Yaskawa INFORM job: OK_R2_O38-47,64(1)(90,180)OKKR.JBI

/JOB
//NAME OK_R2_O38-47,64(1)(90,180)OKKR
///FOLDERNAME X4
//POS
///NPOS 675,675,675,19,0,0
///TOOL 0
///POSTYPE PULSE
///PULSE
C00000=-90909,-97924,-91406,-33882,56334,85304
C00001=-91259,-96225,-90754,-33542,56592,85046
C00002=-84346,-10282,-49110,5038,88729,85099
C00003=-80520,72534,46153,-179,119568,81737
C00004=-84341,50404,17488,-7249,115666,79799
C00005=-84629,52012,20689,-7225,114506,79766
C00006=-84629,51890,21633,-7182,113865,79809
C00007=-84629,52012,20689,-7225,114506,79766
C00008=-84940,55701,25098,-7229,113667,79705
C00009=-84940,55628,25812,-7200,113194,79735
C00010=-84829,53963,24073,-7195,113413,79762
C00011=-84779,55348,25092,-7189,113502,79775
C00012=-83953,58737,25467,-6224,116924,79977
C00013=-84346,-10282,-49110,5038,88729,85099
C00014=-83106,-20728,-52489,-22212,92643,80661
C00015=-106659,-18282,-50653,-15937,87636,73637
C00016=-135463,84611,26036,-8427,98138,63561
C00017=-134711,78652,30015,-19475,126025,58919
C00018=-134415,83458,36943,-18891,124399,59387
C00019=-134415,83178,37391,-18788,124001,59464
C00020=-134415,82845,37969,-18663,123504,59559
C00021=-134415,83107,37513,-18763,123898,59484
C00022=-133823,86478,41707,-18417,123218,59859
C00023=-133823,86166,42311,-18294,122713,59953
C00024=-134051,84793,40603,-18428,122994,59806
C00025=-133823,86534,41603,-18437,123307,59843
C00026=-130836,86678,38865,-21284,122414,55409
C00027=-135463,84611,26036,-8427,98138,63561
C00028=-106659,-18282,-50653,-15937,87636,73637
C00029=-89310,-122172,-106686,-13361,50676,45199
C00030=-123165,-113898,-119110,19125,43336,-19368
C00031=-123668,-102412,-109547,19577,43467,-19587
C00032=-131184,63359,57441,15233,67840,-18691
C00033=-122068,78147,74274,12505,69533,-15106
C00034=-122051,87849,89370,12875,65325,-15559
C00035=-122051,89227,92048,12969,64408,-15664
C00036=-122316,85057,86118,12868,65923,-15592
C00037=-122667,82911,83414,12880,66527,-15655
C00038=-122667,83831,85320,12946,65844,-15732
C00039=-122426,86931,89254,12983,65000,-15737
C00040=-122963,79390,78884,12845,67528,-15654
C00041=-130632,64185,60223,15235,66493,-18662
C00042=-131662,58983,54996,15425,67212,-18954
C00043=-131668,55339,42428,14901,72880,-18222
C00044=-146861,-92393,-105699,36485,53490,-27620
C00045=-148000,-101656,-114811,36865,54640,-27702
C00046=-148000,-101656,-114811,36865,54640,-27702
C00047=-148000,-101656,-114811,36865,54640,-27702
C00048=-159496,-161049,-136264,30615,73499,-21221
C00049=-103228,-122632,-133352,-7038,92284,-523
C00050=-103228,-122632,-133352,-7038,92284,-523
C00051=-103228,-124480,-131601,-7026,90271,-411
C00052=-103391,-121920,-131082,-6996,91247,-517
C00053=-103853,-115329,-128981,-6922,93290,-780
C00054=-103391,-120798,-132087,-7006,92433,-583
C00055=-104641,-114737,-130152,-6774,94243,-1084
C00056=-104641,-114737,-130152,-6774,94243,-1084
C00057=-104641,-116137,-129119,-6762,92896,-1012
C00058=-104641,-115940,-129279,-6764,93095,-1023
C00059=-105111,-108950,-126961,-6694,95208,-1287
C00060=-104576,-115792,-130426,-6785,93876,-1044
C00061=-103741,-127928,-135528,-6927,90867,-609
C00062=-103741,-127928,-135528,-6927,90867,-609
C00063=-103741,-127928,-135528,-6927,90867,-609
C00064=-103865,-116944,-129962,-6921,93061,-771
C00065=-103865,-118485,-128547,-6909,91408,-679
C00066=-103865,-118011,-129031,-6913,91946,-709
C00067=-104350,-111197,-126797,-6823,94018,-978
C00068=-103645,-119716,-131347,-6963,92509,-670
C00069=-126331,-111187,-127566,-2170,93341,-7936
C00070=-126314,-110675,-127191,-2173,93374,-7931
C00071=-126314,-111741,-126360,-2171,92316,-7913
C00072=-126314,-111248,-126762,-2172,92816,-7922
C00073=-126152,-104604,-124481,-2216,94828,-7909
C00074=-126314,-111061,-126906,-2173,93001,-7925
C00075=-125902,-111149,-126935,-2263,92984,-7794
C00076=-132196,-109284,-126305,2386,93568,-14490
C00077=-132014,-110397,-125220,2342,92324,-14457
C00078=-132014,-111538,-124094,2340,91046,-14481
C00079=-132014,-110972,-124684,2340,91699,-14468
C00080=-131346,-109003,-124013,2196,92280,-14246
C00081=-132122,-112463,-125993,2364,91740,-14502
C00082=-130696,-128652,-136015,2037,89553,-14081
C00083=-130696,-128652,-136015,2037,89553,-14081
C00084=-134573,-129962,-127961,2886,84044,-15460
C00085=-135247,-123905,-124729,3029,85191,-15657
C00086=-135247,-124242,-122895,3032,83891,-15687
C00087=-135059,-121526,-122583,2986,85086,-15595
C00088=-134621,-115318,-120572,2888,87018,-15405
C00089=-135273,-124345,-124575,3033,84868,-15671
C00090=-101634,-140552,-130463,-4330,80438,-4385
C00091=-100831,-135445,-127742,-4507,81431,-4148
C00092=-100831,-135220,-126147,-4516,80567,-4118
C00093=-100831,-135304,-126661,-4513,80840,-4129
C00094=-101541,-127818,-124438,-4340,83274,-4455
C00095=-100689,-136992,-128168,-4541,80909,-4084
C00096=-101700,-117063,-135109,-4321,95328,-4920
C00097=-101700,-117063,-135109,-4321,95328,-4920
C00098=-107464,-106510,-121453,-3057,92107,-6652
C00099=-105693,-105772,-119256,-3437,91202,-6062
C00100=-105693,-106748,-117862,-3435,89847,-6024
C00101=-105693,-106325,-118509,-3436,90460,-6041
C00102=-104724,-99451,-116018,-3652,92493,-5788
C00103=-105563,-106984,-120499,-3466,91350,-6023
C00104=-97637,-124436,-133710,-5150,90918,-3458
C00105=-101700,-117063,-135109,-4321,95328,-4920
C00106=-101700,-117063,-135109,-4321,95328,-4920
C00107=-113885,-115939,-123860,-1658,88568,-8649
C00108=-113885,-115976,-123799,-1658,88510,-8649
C00109=-113885,-116503,-122835,-1658,87648,-8639
C00110=-113928,-115223,-122529,-1647,88114,-8658
C00111=-114061,-111130,-121156,-1620,89368,-8717
C00112=-113613,-117192,-124203,-1715,88138,-8556
C00113=-77135,-109099,-124316,-9289,94737,2930
C00114=-77964,-100968,-118468,-9143,95217,2626
C00115=-77964,-101677,-117713,-9127,94398,2685
C00116=-77964,-101560,-117850,-9129,94540,2675
C00117=-78928,-97543,-116360,-8967,95572,2290
C00118=-77908,-100245,-119438,-9173,96179,2574
C00119=-71973,-123086,-130703,-10190,92110,4818
C00120=-61369,-106979,-129386,18745,110548,-43775
C00121=-54050,-118433,-122678,29834,105379,-66043
C00122=-54050,-118432,-122677,29849,105379,-66042
C00123=-52380,-128849,-120518,29019,98947,-67079
C00124=-52380,-128559,-118965,28945,98241,-67262
C00125=-52380,-128751,-119946,28990,98681,-67146
C00126=-50245,-132811,-121152,28917,96763,-66805
C00127=-52380,-128751,-119946,28990,98681,-67146
C00128=-49374,-119498,-117890,29381,100712,-65454
C00129=-49135,-119946,-117683,29342,100317,-65463
C00130=-49135,-119959,-116418,29258,99629,-65643
C00131=-49135,-119963,-116925,29289,99902,-65571
C00132=-47420,-122909,-117861,29192,98489,-65269
C00133=-49767,-118756,-118042,29437,101266,-65461
C00134=-58824,-127197,-127906,29549,105900,-67783
C00135=-58824,-127197,-127906,29549,105900,-67783
C00136=-55789,-138532,-125635,28743,98511,-68512
C00137=-54845,-137144,-123724,28738,97781,-68329
C00138=-54845,-136558,-122036,28679,97131,-68490
C00139=-54845,-136878,-122937,28709,97474,-68406
C00140=-52687,-141381,-124200,28678,95380,-68093
C00141=-56052,-135036,-125386,28893,100051,-68223
C00142=-56052,-135036,-125386,28893,100051,-68223
C00143=-54923,-136926,-123517,28734,97796,-68355
C00144=-54923,-136449,-122129,28684,97260,-68488
C00145=-54923,-136715,-122887,28711,97551,-68416
C00146=-52628,-141500,-124230,28677,95326,-68085
C00147=-54923,-138669,-131970,29176,101590,-67387
C00148=-49576,-128334,-132403,27234,106270,-69223
C00149=-44922,-139442,-128392,26353,97465,-69516
C00150=-43106,-142181,-127565,26251,95168,-69348
C00151=-43106,-141292,-125343,26201,94348,-69532
C00152=-43106,-141708,-126356,26223,94717,-69449
C00153=-42222,-150085,-128620,26118,91814,-69764
C00154=-43106,-141708,-126356,26223,94717,-69449
C00155=-58006,-149727,-131155,24086,101568,-78058
C00156=-67130,-160484,-130477,19696,102779,-86761
C00157=-65656,-163702,-131169,20680,100336,-85246
C00158=-25743,-109032,-115433,27145,106620,-70118
C00159=-31386,-185321,-134069,30256,67850,-60806
C00160=-40913,-181249,-136978,30366,76641,-63974
C00161=-31337,-124593,-132531,25311,107075,-53461
C00162=-107165,-96970,-126665,-3187,100215,-6761
C00163=-107165,-106401,-121090,-3121,91950,-6553
C00164=-99006,-123912,-120398,-10471,76789,317
C00165=-104449,-120133,-119195,-8811,77334,-1598
C00166=-136314,-76901,-102772,1273,87959,-12257
C00167=-129245,-75238,-102051,-6216,89043,-4909
C00168=-138081,-104464,-122106,1833,85725,-12838
C00169=-119260,-105046,-123410,-8534,87528,-2432
C00170=-124620,-151805,-134891,-7305,72242,-3267
C00171=-124614,-151414,-134787,-7302,72378,-3273
C00172=-124612,-151215,-134734,-7300,72449,-3276
C00173=-124620,-151805,-134891,-7305,72242,-3267
C00174=-127969,-108981,-129625,-6073,90620,-5362
C00175=-128058,-112032,-130642,-6044,89675,-5344
C00176=-99990,-117497,-120264,-13536,83880,4252
C00177=-95946,-115412,-117807,-14495,84133,5598
C00178=-139069,-101671,-113062,-2900,83618,-8638
C00179=-134512,-124069,-125019,-4259,79673,-7022
C00180=-124704,-125859,-130096,-7035,82535,-3892
C00181=-99313,-127153,-133045,12119,95446,-32872
C00182=-57886,-133831,-130402,29291,103936,-67934
C00183=-55789,-138532,-125635,28743,98511,-68512
C00184=-48693,-117877,-116324,29063,104784,-69163
C00185=-50073,-120833,-117390,28223,106210,-71565
C00186=-68626,-163926,-129258,19114,104295,-87122
C00187=-70376,-133538,-127464,20847,118406,-85282
C00188=-70376,-133538,-127464,20847,118406,-85282
C00189=-57461,-97931,-109353,30188,105270,-63675
C00190=-56121,-79134,-101591,31100,116741,-68778
C00191=-90239,-137211,-122130,21625,111934,-84005
C00192=-78206,-119593,-116830,16675,122083,-90308
C00193=-77714,-101700,-117389,19308,131076,-88387
C00194=-81561,-124200,-134149,21063,125175,-90603
C00195=-103376,-109759,-132308,-3968,97270,-5504
C00196=-101634,-140552,-130463,-4330,80438,-4385
C00197=-110031,-125673,-123303,3182,83425,-15942
C00198=-90641,-116743,-120449,-11075,89773,6751
C00199=-125358,-116095,-120243,-4332,86705,-4548
C00200=-114606,-95150,-113030,-13927,98680,11559
C00201=-109678,-119625,-133746,-14623,99658,13079
C00202=-112326,-124641,-135293,-14185,97639,12436
C00203=-113675,-111285,-124420,-14007,97585,11993
C00204=-113699,-111426,-124467,-14002,97539,11990
C00205=-124004,-129907,-130136,-8507,87303,2218
C00206=-139409,-131326,-130615,456,84743,-11777
C00207=-149006,-99791,-120232,2566,94725,-14751
C00208=-149042,-99754,-120218,2574,94737,-14762
C00209=-144445,-99331,-120062,1565,94748,-13320
C00210=-148134,-92536,-117492,2386,96740,-14437
C00211=-154718,-145008,-134516,3815,80522,-16974
C00212=-155631,-143491,-134098,4008,81086,-17267
C00213=-124045,-119827,-121338,-6126,86009,-1689
C00214=-127884,-116949,-120404,-5328,86643,-2988
C00215=-148100,-95243,-112662,-980,92257,-9671
C00216=-137287,-91556,-109748,-13625,92659,296
C00217=-127829,-127486,-128792,-15513,87749,4031
C00218=-127829,-122446,-134816,-15592,93826,3264
C00219=-125285,-108995,-105645,24533,66859,-22374
C00220=-121876,-100663,-100590,22961,66967,-21017
C00221=-120611,-97454,-98556,22372,66992,-20522
C00222=-120728,-95778,-96365,22498,66572,-20652
C00223=-120611,-97454,-98556,22372,66992,-20522
C00224=-120972,-98646,-98782,22597,66650,-20731
C00225=-119814,-94892,-97816,21908,67582,-20099
C00226=-120972,-98646,-98782,22597,66650,-20731
C00227=-122255,-101873,-100811,23195,66623,-21236
C00228=-125713,-110249,-105850,24792,66512,-22621
C00229=-125414,-109454,-110952,25434,70557,-21724
C00230=-121886,-100912,-105844,23885,70668,-20357
C00231=-120575,-97642,-103795,23303,70688,-19860
C00232=-120636,-96154,-101667,23400,70203,-19982
C00233=-120575,-97642,-103795,23303,70688,-19860
C00234=-121028,-97980,-103315,23548,70382,-20093
C00235=-119871,-93906,-102218,22897,71374,-19458
C00236=-121028,-97980,-103315,23548,70382,-20093
C00237=-122351,-101230,-105354,24132,70373,-20595
C00238=-125908,-109706,-110431,25687,70298,-21973
C00239=-125468,-108852,-114009,26132,73198,-21211
C00240=-121864,-100250,-108878,24604,73277,-19846
C00241=-120523,-96969,-106822,24029,73283,-19350
C00242=-120543,-95651,-104748,24106,72739,-19471
C00243=-120523,-96969,-106822,24029,73283,-19350
C00244=-121096,-97384,-106424,24308,73024,-19616
C00245=-119937,-93066,-105230,23683,74062,-18974
C00246=-121096,-97384,-106424,24308,73024,-19616
C00247=-122450,-100644,-108468,24886,73032,-20117
C00248=-126090,-109173,-113564,26418,72994,-21493
C00249=-126107,-105383,-120588,25792,78658,-20214
C00250=-115870,-101424,-121533,-41206,90180,-3452
C00251=-115851,-106682,-115012,-41260,85065,-1433
C00252=-119242,-98694,-109765,-40357,84214,-2540
C00253=-120508,-95652,-107669,-40003,83867,-2939
C00254=-120512,-93942,-105232,-40036,83383,-2757
C00255=-120508,-95652,-107669,-40003,83867,-2939
C00256=-119976,-95300,-106376,-40178,83625,-2624
C00257=-123146,-93912,-105979,-39274,82602,-3565
C00258=-119976,-95300,-106376,-40178,83625,-2624
C00259=-118706,-98291,-108457,-40527,83992,-2228
C00260=-115305,-106116,-113657,-41413,84900,-1133
C00261=-117529,-113204,-110114,-15038,59483,16836
C00262=-119860,-102582,-104476,-13511,61010,15725
C00263=-120710,-98611,-102232,-12973,61516,15338
C00264=-120712,-96036,-99318,-13028,61058,15391
C00265=-120710,-98611,-102232,-12973,61516,15338
C00266=-120133,-97446,-101425,-13271,61707,15536
C00267=-121539,-92419,-99938,-12330,63118,14842
C00268=-120133,-97446,-101425,-13271,61707,15536
C00269=-119274,-101350,-103659,-13810,61233,15923
C00270=-116924,-111770,-109266,-15331,59803,17031
C00271=-118012,-90030,-113480,-10859,76824,11039
C00272=-121151,-43618,-104634,1145,105190,-4571
C00273=-120753,-40362,-99446,1000,103667,-4481
C00274=-120604,-39041,-97355,946,103057,-4446
C00275=-120606,-40163,-95662,941,101440,-4458
C00276=-120604,-39041,-97355,946,103057,-4446
C00277=-120772,-35445,-95769,1008,103931,-4483
C00278=-120462,-29091,-92658,908,105279,-4391
C00279=-120772,-35445,-95769,1008,103931,-4483
C00280=-120921,-36668,-97839,1062,104577,-4517
C00281=-121319,-39651,-102962,1210,106200,-4605
C00282=-108629,-121399,-122702,-16889,67135,14241
C00283=-115336,-113367,-105488,-19088,53546,18271
C00284=-117865,-102996,-100223,-17109,54980,16930
C00285=-118786,-99066,-98108,-16412,55481,16461
C00286=-118815,-96798,-95161,-16518,54853,16552
C00287=-118786,-99066,-98108,-16412,55481,16461
C00288=-119112,-97264,-98148,-16039,56331,16193
C00289=-118757,-93015,-97035,-15990,57843,16106
C00290=-119112,-97264,-98148,-16039,56331,16193
C00291=-123316,-98367,-98161,-13561,55035,14648
C00292=-126858,-97217,-97820,-11275,54872,13210
C00293=-123316,-98367,-98161,-13561,55035,14648
C00294=-122519,-102389,-100318,-14180,54451,15058
C00295=-120328,-113051,-105701,-15959,52759,16243
C00296=-124093,-110707,-95637,16539,52225,-18162
C00297=-121727,-101468,-90458,14864,53273,-16967
C00298=-120864,-97923,-88367,14268,53637,-16545
C00299=-120864,-95769,-85768,14357,53158,-16613
C00300=-120864,-97923,-88367,14268,53637,-16545
C00301=-120753,-94948,-87925,13988,54838,-16331
C00302=-119636,-91806,-87160,13170,55764,-15745
C00303=-120753,-94948,-87925,13988,54838,-16331
C00304=-121593,-98445,-90034,14553,54501,-16732
C00305=-123889,-107558,-95262,16133,53518,-17861
C00306=-123907,-109460,-104253,15319,57915,-17198
C00307=-120718,-89127,-94408,-93,103364,81793
C00308=-120702,-88967,-86044,-90,98299,81802
C00309=-120714,-92346,-83648,-90,95088,81800
C00310=-120719,-93530,-82604,-90,93837,81800
C00311=-120721,-91291,-79709,-90,93204,81799
C00312=-120719,-93530,-82604,-90,93837,81800
C00313=-120503,-94372,-82680,-81,93451,81873
C00314=-120503,-97134,-83277,-81,92401,81874
C00315=-120503,-94372,-82680,-81,93451,81873
C00316=-120501,-93212,-83739,-81,94699,81873
C00317=-120496,-89894,-86173,-82,97902,81873
C00318=-120512,-90208,-94601,-84,102927,81864
C00319=-120739,-87258,-85833,-92,99047,81789
C00320=-120752,-90752,-83510,-91,95822,81787
C00321=-120758,-91982,-82493,-91,94564,81786
C00322=-120759,-89478,-79257,-91,93861,81786
C00323=-120758,-91982,-82493,-91,94564,81786
C00324=-120462,-95334,-83503,-80,93464,81887
C00325=-120461,-97919,-84058,-79,92477,81888
C00326=-120462,-95334,-83503,-80,93464,81887
C00327=-120460,-94163,-84562,-80,94717,81887
C00328=-120456,-90813,-86994,-80,97935,81887
C00329=-121033,-93279,-128320,140,99068,-4698
C00330=-120997,-110061,-117241,128,83627,-4703
C00331=-120579,-101211,-110995,15,84330,-4566
C00332=-120424,-97983,-108548,-25,84483,-4515
C00333=-120430,-96385,-106046,-24,83763,-4517
C00334=-120424,-97983,-108548,-25,84483,-4515
C00335=-120936,-92390,-106244,111,85940,-4681
C00336=-120538,-86818,-104536,4,87751,-4552
C00337=-120936,-92390,-106244,111,85940,-4681
C00338=-121096,-95373,-108656,154,85891,-4732
C00339=-121527,-103462,-114785,270,85508,-4872
C00340=-75677,-91018,-121004,-38809,104477,-3256
C00341=-86494,-89564,-122641,-29897,102391,-4704
C00342=-121241,-108971,-117698,1136,79653,-4828
C00343=-120728,-99263,-111358,963,80734,-4651
C00344=-120539,-95742,-108880,900,81016,-4587
C00345=-120543,-94296,-106552,902,80326,-4593
C00346=-120539,-95742,-108880,900,81016,-4587
C00347=-120728,-93992,-107595,961,81127,-4647
C00348=-120728,-90301,-106424,959,82303,-4638
C00349=-120728,-93992,-107595,961,81127,-4647
C00350=-121024,-97533,-112143,1058,82109,-4735
C00351=-121551,-107098,-118478,1235,81100,-4915
C00352=-121569,-100080,-124444,1231,88376,-4850
C00353=-117898,-83225,-110918,-12916,113641,67504
C00354=-119870,-90654,-110250,-12481,109228,67312
C00355=-120686,-93336,-109842,-12338,107519,67211
C00356=-120688,-92183,-107571,-12276,106730,67294
C00357=-120686,-93336,-109842,-12338,107519,67211
C00358=-120163,-91649,-109473,-12395,108219,67318
C00359=-121681,-97188,-111137,-12239,106219,67001
C00360=-120163,-91649,-109473,-12395,108219,67318
C00361=-119359,-88923,-109851,-12543,109932,67413
C00362=-117416,-81399,-110449,-12994,114344,67589
C00363=-120617,-94125,-108136,8857,121741,88541
C00364=-120616,-94449,-107526,8800,121205,88496
C00365=-136098,-107181,-107429,16269,112846,84409
C00366=-120444,-95183,-107742,8816,120947,88541
C00367=-119761,-91680,-105499,9024,121288,-74873
C00368=-120616,-95784,-105179,-19399,105655,65758
C00369=-120617,-94769,-108163,-19676,107886,65380
C00370=-121686,-93853,-106574,-24019,104588,57765
C00371=-120617,-92780,-110041,-24421,107344,57569
C00372=-120617,-90665,-112384,-24828,109654,57058
C00373=-120619,-82046,-117525,-26421,116533,55408
C00374=-120645,-81988,-112872,-3577,88664,15070
C00375=-120614,-96077,-90479,12976,48732,-14983
C00376=-120612,-93911,-81283,13967,44304,-15634
C00377=-120612,-93390,-79613,14157,43566,-15753
C00378=-121252,-93346,-79166,14714,43437,-16096
C00379=-121500,-95247,-79374,15137,42660,-16355
C00380=-120782,-94947,-80724,14317,43483,-15851
C00381=-120611,-93982,-79716,14233,43318,-15795
C00382=-120612,-95725,-83890,13821,44941,-15536
C00383=-121326,-94847,-83951,14224,45559,-15784
C00384=-120613,-94980,-84633,13612,45776,-15407
C00385=-120613,-95388,-86250,13438,46540,-15293
C00386=-120616,-96933,-104006,-5046,49827,-739
C00387=-120616,-97132,-103061,-5097,49146,-704
C00388=-120617,-95323,-101728,-5088,49256,-711
C00389=-120871,-100699,-104338,-4972,48087,-759
C00390=-120795,-98262,-101888,-5054,47837,-712
C00391=-120618,-95198,-103493,-5003,50401,-770
C00392=-121122,-95129,-103646,-4600,50501,-986
C00393=-120617,-97030,-104927,-5009,50342,-766
C00394=-120617,-96757,-105844,-4959,51045,-801
C00395=-120618,-92718,-112658,-4589,57292,-1090
C00396=-108098,-105677,-132023,-7461,89264,328
C00397=-80455,-75739,-120669,-16714,100968,7375
C00398=-97258,-84752,-105297,-10869,90674,3530
C00399=-97358,-86422,-102930,-10833,88387,3696
C00400=-97424,-86715,-102018,-10818,87679,3736
C00401=-97216,-90521,-102980,-10875,86365,3919
C00402=-97404,-84940,-102216,-10822,88698,3655
C00403=-120617,-94266,-106774,-4665,84598,-3614
C00404=-111454,-84543,-103018,-13521,90962,7073
C00405=-109783,-86139,-104921,-12729,90791,5985
C00406=-106092,-100123,-116923,-13597,91547,7106
C00407=-102052,-116072,-128299,-14497,91044,8487
C00408=-91007,-121504,-125767,-15485,91359,21712
C00409=-120613,-95050,-86060,-3557,95049,80550
C00410=-120612,-93945,-81838,-3544,93023,80607
C00411=-121155,-91942,-79314,-3616,92478,80448
C00412=-120652,-94806,-81837,-3543,92579,80606
C00413=-120610,-90975,-79567,-3544,93151,80605
C00414=-150255,-82598,-75582,-4413,93505,70504
C00415=-122384,-91795,-77981,-11848,92227,69969
C00416=-120612,-93489,-79991,-12120,92904,70125
C00417=-120613,-94640,-84016,-12161,94749,69944
C00418=-120614,-96377,-93023,-12320,99298,69491
C00419=-120644,-125570,-121052,6784,67869,5403
C00420=-120615,-96622,-98748,12572,58745,-14095
C00421=-120615,-96643,-96984,12717,57674,-14222
C00422=-127606,-89142,-93330,20657,62312,-19456
C00423=-120926,-99715,-97034,13118,56212,-14526
C00424=-120613,-97817,-97899,12721,57634,-14225
C00425=-120615,-96818,-95655,-6616,54391,-866
C00426=-120615,-97044,-96976,-6561,55085,-910
C00427=-112093,-90513,-93108,-22044,58833,17349
C00428=-120615,-96644,-96112,-9528,53512,9485
C00429=-120615,-96653,-97679,-9416,54459,9397
C00430=-120616,-95373,-105489,-8868,59856,8934
C00431=-117333,-91440,-108817,-14098,83709,30265
C00432=-112347,-94381,-87846,-22750,99580,64599
C00433=-112329,-92021,-78548,-22454,95406,65402
C00434=-115628,-91274,-75119,-22621,92902,64661
C00435=-117255,-90241,-73175,-22718,91835,64269
C00436=-117028,-88603,-73220,-22719,92705,64185
C00437=-116923,-92272,-75451,-22697,92259,64308
C00438=-120553,-90828,-77383,15099,94128,70510
C00439=-120613,-90885,-77384,15804,94030,70628
C00440=-123770,-105111,-82751,16580,84167,79857
C00441=-124886,-104010,-85216,16560,86394,79763
C00442=-120613,-94284,-84162,15892,96365,70931
C00443=-120614,-95920,-93129,16139,100869,71526
C00444=-120649,-92160,-111225,3199,84919,49711
C00445=-120616,-97604,-99172,-11891,40402,23254
C00446=-120614,-96911,-90603,-13253,35598,24030
C00447=-120614,-96763,-89737,-13401,35153,24111
C00448=-121291,-96342,-89250,-12683,34963,23744
C00449=-119113,-97762,-90324,-15090,35268,24978
C00450=-120705,-99580,-90146,-13704,33974,24279
C00451=-121588,-95238,-86691,-12692,33949,23762
C00452=-127502,-77730,-88040,1756,56127,19882
C00453=-125086,-93679,-98074,150,54079,20822
C00454=-120613,-95818,-85653,-14108,33181,24494
C00455=-120615,-97479,-97669,-6545,55280,-923
C00456=-121580,-96410,-96097,-5967,54791,-1285
C00457=-120928,-100587,-97757,-6468,53722,-953
C00458=-120613,-98670,-98620,-6548,55254,-920
C00459=-120615,-96854,-96360,-6584,54805,-893
C00460=-120615,-97074,-97513,-6537,55399,-931
C00461=-114077,-92170,-94328,-19163,57465,15491
C00462=-120615,-97626,-97578,-9481,53904,9448
C00463=-120636,-112691,-117418,-8831,59265,10492
C00464=-120617,-94408,-109491,-7961,65698,13071
C00465=-120616,-97035,-102174,-8375,59902,13490
C00466=-120616,-97254,-100452,-8474,58742,13580
C00467=-120616,-96110,-99125,-8495,58514,13598
C00468=-120614,-98453,-101360,-8481,58685,13585
C00469=-119727,-100186,-100479,-9138,57364,14041
C00470=-120617,-96158,-99373,-8483,58642,13587
C00471=-120616,-97215,-100721,-8458,58926,13566
C00472=-120616,-96978,-102436,-8360,60091,13476
C00473=-120617,-94247,-109716,-7948,65917,13056
C00474=-120616,-96445,-103082,5252,59171,-13430
C00475=-120615,-96888,-94956,5569,53965,-13694
C00476=-120614,-96711,-93127,5642,52935,-13750
C00477=-120614,-96618,-92386,5672,52529,-13773
C00478=-119756,-94067,-91753,5051,53390,-13370
C00479=-120525,-97964,-94062,5589,52861,-13717
C00480=-120614,-96681,-92800,5656,52750,-13760
C00481=-120614,-96709,-92988,5648,52851,-13755
C00482=-120614,-96767,-93400,5632,53074,-13742
C00483=-120614,-96843,-94134,5603,53484,-13720
C00484=-120615,-96977,-95945,5531,54526,-13664
C00485=-120616,-97003,-101109,6851,58481,-13557
C00486=-120615,-97139,-99377,6934,57353,-13629
C00487=-120615,-97164,-98672,6968,56909,-13657
C00488=-119756,-94335,-97933,6375,57832,-13263
C00489=-120570,-98373,-100300,6912,57283,-13615
C00490=-120615,-97165,-99156,6946,57204,-13638
C00491=-120616,-97129,-99856,6912,57651,-13610
C00492=-120616,-96964,-101578,6829,58787,-13537
C00493=-120617,-96349,-105255,7716,61917,-13386
C00494=-120616,-96771,-103611,7804,60699,-13471
C00495=-120616,-96905,-102940,7840,60222,-13505
C00496=-119756,-93851,-102113,7266,61195,-13116
C00497=-120602,-97980,-104523,7800,60639,-13470
C00498=-120616,-96844,-103353,7819,60505,-13485
C00499=-120616,-96699,-104019,7783,60985,-13451
C00500=-120617,-96245,-105652,7696,62212,-13366
C00501=-120618,-92150,-112439,7334,68442,-12961
C00502=-130920,-122289,-127601,-23263,76296,33617
C00503=-126647,-121486,-124764,-14921,71090,19914
C00504=-118673,-117816,-113052,-9081,54805,1270
C00505=-119719,-97166,-102733,-8035,58912,525
C00506=-118944,-92090,-109805,-27006,83902,36269
C00507=-120616,-93914,-111601,-26462,83549,35758
C00508=-120617,-94475,-108119,-24525,75199,30020
C00509=-120618,-90011,-113520,-23738,94905,43572
C00510=-120617,-93534,-109718,-22404,79768,31867
C00511=-120617,-93028,-110386,-24696,84592,28860
C00512=-120617,-93859,-109223,-24523,82429,27907
C00513=-120617,-95217,-106728,-22357,73913,21133
C00514=-120616,-96198,-104144,-16550,64688,11231
C00515=-120616,-97587,-102867,-7505,58697,196
C00516=-120615,-98378,-102979,677,57412,-8649
C00517=-120615,-98092,-104435,2505,58558,-10610
C00518=-120615,-97859,-104607,2041,58746,-10113
C00519=-120615,-97689,-104685,1580,58853,-9618
C00520=-120615,-97267,-104663,-2078,59079,-5700
C00521=-122185,-96113,-104438,-1107,59504,-6297
C00522=-124417,-94235,-103728,259,60020,-7133
C00523=-120617,-96195,-105273,-2057,60007,-5718
C00524=-120617,-95777,-106468,-2039,60956,-5736
C00525=-120690,-30346,-78642,22937,64170,-21118
C00526=-120690,-30346,-78642,22937,64170,-21118
C00527=-98469,-5770,-79404,6171,73775,-13621
C00528=-73961,-64832,-115099,-11040,66386,-6438
C00529=-152983,-151482,-105999,63266,53723,19798
C00530=-133395,-32083,-56059,41211,61963,37621
C00531=-138234,23065,45169,67508,45202,44915
C00532=-136781,30072,55747,70235,43147,43411
C00533=-136213,33214,60449,71542,42329,42699
C00534=-136213,31591,57334,70422,42710,43384
C00535=-136788,30891,57778,71075,42855,42892
C00536=-134893,29619,56778,71118,41623,43172
C00537=-133284,25640,52793,70642,40733,43707
C00538=-131869,22445,49655,70246,39929,44150
C00539=-132436,19576,45433,69035,40713,44782
C00540=-133889,13007,35719,66469,42691,46136
C00541=-120930,8852,32410,71146,24358,44597
C00542=-120056,16713,42856,76185,23038,42237
C00543=-120570,20810,47735,78353,23157,41125
C00544=-120179,17981,45384,78314,22894,41190
C00545=-119718,18730,44666,76295,22791,42223
C00546=-125399,29317,56132,80433,26238,39500
C00547=-125034,24898,50699,78244,26224,40637
C00548=-126001,16678,39521,73266,27604,43020
C00549=-110893,28996,24386,6920,61269,70362
C00550=-121937,-147756,-98721,13314,47766,64479
C00551=-71720,-152863,-104081,-12596,70757,83485
C00552=-71720,-152863,-104081,-12596,70757,83485
C00553=-91982,-28216,-51992,2303,92813,79298
C00554=-105745,54824,-16277,12342,106777,76346
C00555=-79811,47197,33770,-5226,114025,80115
C00556=-80023,42119,31306,-5246,112923,80086
C00557=-80397,41231,31844,-5317,112121,79984
C00558=-80109,39795,28796,-5290,113266,80037
C00559=-80112,42618,33014,-5241,112126,80089
C00560=-81014,41143,31800,-5517,112061,79755
C00561=-81200,40698,29696,-5625,113108,79635
C00562=-82013,41869,30925,-5879,112897,79339
C00563=-84094,42448,33219,-3257,112240,82331
C00564=-82696,41301,31992,-6274,111848,78881
C00565=-83189,43833,33118,-6256,112463,78920
C00566=-80599,47195,33767,-5484,113974,79819
C00567=-80608,45992,24153,-5781,119246,79546
C00568=-80156,46426,18785,-6968,101557,41119
C00569=-78753,47274,23775,-10662,32517,-78562
C00570=-79428,-41610,-51646,-9616,33163,-79071
C00571=-79413,-40970,-42943,-11157,28217,-78271
C00572=-79779,-35257,-36372,-11029,27079,-78324
C00573=-80609,-32957,-33621,-9964,26475,-78835
C00574=-79917,-33213,-35108,-10725,27328,-78472
C00575=-79914,-35155,-35130,-11097,26361,-78286
C00576=-81360,-33165,-33796,-8816,26388,-79388
C00577=-81501,-33436,-35517,-8333,27283,-79626
C00578=-82704,-33725,-35707,-6541,27141,-80488
C00579=-82488,-32797,-33501,-7076,26287,-80226
C00580=-83572,-32639,-33468,-5384,26265,-81042
C00581=-83984,-33203,-37030,-4447,28135,-81499
C00582=-80764,-40975,-42948,-9214,28047,-79206
C00583=-80778,-41615,-51650,-7929,33019,-79872
C00584=-83330,-46575,-52890,-13958,55049,-41505
C00585=-86193,-52033,-54165,-20785,79907,1804
C00586=-87571,-35325,-52921,-25788,81678,348
C00587=-87508,-34952,-39783,-27132,74543,196
C00588=-104644,32154,27534,4448,60513,72731
C00589=-93805,201,18674,23355,11914,69008
C00590=-93808,216,18686,23365,11915,69004
C00591=-93810,222,18691,23369,11915,69002
C00592=-93638,2355,20486,22861,11860,69245
C00593=-93955,-2017,16089,22978,12371,69170
C00594=-93808,210,18682,23363,11914,69005
C00595=-93806,198,18671,23357,11914,69008
C00596=-93804,186,18662,23351,11913,69011
C00597=-93802,180,18657,23347,11913,69012
C00598=-93799,166,18644,23338,11912,69017
C00599=-93810,232,18700,23265,11906,69051
C00600=-93813,246,18712,23275,11907,69047
C00601=-94451,684,18996,25087,12134,68175
C00602=-93990,-1863,16961,23823,11950,68785
C00603=-93814,-607,16661,21825,12670,69707
C00604=-100120,3293,21094,39224,14315,61321
C00605=-100936,-4761,10472,35572,16592,62958
C00606=-101724,-18723,-6868,31140,19848,65000
C00607=-104644,32154,27534,4448,60513,72731
C00608=-81813,-56841,-53371,-53266,50302,14082
C00609=-60380,-131230,-84967,-114894,34586,40161
C00610=-75788,-111312,-115723,-41491,75595,63087
C00611=-90161,-54224,-109841,7916,106787,80704
C00612=-89492,4607,-58591,7657,105439,80800
C00613=-89900,18802,-35938,9766,95357,80687
C00614=-83481,65005,13429,-9056,119285,78997
C00615=-83912,59570,13434,-8836,116477,79073
C00616=-105122,63991,30490,2309,126100,76457
C00617=-105343,61862,26796,2259,127285,76391
C00618=-85790,59910,13822,-8992,116222,78417
C00619=-84859,64061,16437,-8959,116837,78702
C00620=-84733,23156,-31643,-6898,102580,79911
C00621=-89806,-37631,-52942,13196,44828,72538
C00622=-94750,-32934,-45091,18174,44929,69862
C00623=-94750,-25149,-34817,18936,42722,69385
C00624=-107305,-33153,-35053,31246,31625,63156
C00625=-107702,-34958,-34985,32523,30946,62498
C00626=-97165,-24114,-34089,20969,43382,68305
C00627=-95242,-30076,-40811,18964,43932,69406
C00628=-95187,-81119,-79791,20309,40550,69551
C00629=-106636,9561,-40732,-8334,61658,77698
C00630=-105745,52807,-15764,12246,105454,76208
C00631=-120157,82254,53851,-8462,118881,68276
C00632=-120764,76019,49190,-8631,118486,68068
C00633=-120545,73220,47168,-8543,118319,68170
C00634=-121013,73553,46157,-8768,119052,67924
C00635=-120677,76096,50452,-8536,117766,68159
C00636=-121226,74586,48871,-8734,117906,67937
C00637=-121277,74331,46343,-8885,119308,67802
C00638=-123087,79936,53120,-9346,117831,67212
C00639=-123276,78435,53420,-9313,116866,67221
C00640=-123824,79710,55035,-9457,116468,67043
C00641=-123162,86054,59807,-9277,116864,67267
C00642=-123114,53430,10385,-1251,116221,68203
C00643=-136323,52272,9545,44589,64919,61463
C00644=-139783,-33179,-13184,69240,48192,46182
C00645=-137611,-28365,-6875,70201,46216,45730
C00646=-136958,-25590,-3634,70647,45579,45500
C00647=-136770,-25555,-2359,71345,45178,45070
C00648=-137559,-27867,-5282,70853,45921,45309
C00649=-131841,-32953,-8633,70743,41902,45928
C00650=-131975,-36416,-12130,70369,42121,46140
C00651=-134147,-41542,-18435,69427,44030,46529
C00652=-141128,-29133,-31085,43489,44991,50173
C00653=-145944,-19375,-16364,60085,47488,49165
C00654=-146184,-15082,-11889,60605,47355,48817
C00655=-146072,-18893,-14822,60688,47208,48761
C00656=-145286,-17068,-12207,60970,46372,48581
C00657=-149932,-5295,-4298,61545,49901,48162
C00658=-146980,-8744,-14162,48811,51872,51880
C00659=-141391,-26070,-33699,44316,51156,54843
C00660=-135350,-43982,-50251,40364,49000,57185
C00661=-135985,2271,-36804,-9338,77862,64370
C00662=-130949,74091,43956,-19987,113167,60546
C00663=-132080,69549,41488,-20064,112128,60294
C00664=-132880,68865,42086,-20096,111257,60142
C00665=-132541,67844,41901,-19973,110951,60327
C00666=-132116,69898,43068,-19947,111372,60417
C00667=-135736,79269,54433,-20274,108439,59549
C00668=-135060,80104,54141,-20241,109178,59676
C00669=-133923,84725,56898,-20139,110093,59949
C00670=-137379,33195,-5040,-12355,95090,61475
C00671=-141075,-6060,-32928,-6165,69436,63043
C00672=-141075,-2977,-40411,-5973,75592,62734
C00673=-125690,-78122,-87562,-13631,67908,68588
C00674=-2173,-78122,-87562,-13631,67908,68588
BC00000=277590,692280,168144
BC00001=277590,750776,168144
BC00002=277590,791707,168144
BC00003=277590,791707,168144
BC00004=274757,787027,149092
BC00005=274757,787027,149092
BC00006=274757,787027,149092
BC00007=274757,787027,149092
BC00008=274757,787027,149092
BC00009=274757,787027,149092
BC00010=274757,787027,149092
BC00011=274757,787027,149092
BC00012=275390,788044,146099
BC00013=277590,791707,168144
BC00014=277590,791707,168144
BC00015=277590,791707,168144
BC00016=337074,760417,53
BC00017=337074,815057,24896
BC00018=337074,815057,53
BC00019=337074,815057,53
BC00020=337074,815057,53
BC00021=337074,815057,53
BC00022=337074,815057,53
BC00023=337074,815057,53
BC00024=337074,815057,53
BC00025=337074,815057,53
BC00026=337074,815057,53
BC00027=337074,780859,53
BC00028=277590,791707,168144
BC00029=277590,719585,168144
BC00030=96859,683802,308578
BC00031=96859,755769,293742
BC00032=128715,819724,308578
BC00033=128715,834124,308578
BC00034=128715,834124,308578
BC00035=128715,834124,308578
BC00036=128715,834124,308578
BC00037=128715,834124,308578
BC00038=128715,834124,308578
BC00039=128715,834124,308578
BC00040=128715,834124,308578
BC00041=128715,819724,308578
BC00042=128715,819724,308578
BC00043=128715,819724,308578
BC00044=128715,755769,293742
BC00045=128715,683802,308578
BC00046=128715,683802,1074810
BC00047=128715,683802,1074810
BC00048=10701,883002,1074810
BC00049=2462,1013180,1073459
BC00050=106,1014076,1058465
BC00051=106,1014076,1058465
BC00052=106,1014076,1058465
BC00053=106,1014076,1058465
BC00054=106,1014076,1058465
BC00055=75740,998026,1061993
BC00056=76500,998506,1056750
BC00057=76500,998506,1056750
BC00058=76500,998506,1056750
BC00059=76500,998506,1056750
BC00060=76500,998506,1056750
BC00061=76500,998506,1056750
BC00062=62326,958870,1056750
BC00063=67570,962518,1021274
BC00064=67570,962518,1021274
BC00065=67570,962518,1021274
BC00066=67570,962518,1021274
BC00067=67570,962518,1021271
BC00068=67570,962518,1021274
BC00069=67570,962518,1021274
BC00070=67570,962518,1021274
BC00071=67570,962518,1021274
BC00072=67570,962518,1021274
BC00073=67570,962518,1021274
BC00074=67570,962518,1021274
BC00075=145480,943896,1073360
BC00076=166821,969292,1072076
BC00077=166821,969292,1072076
BC00078=166821,969292,1072076
BC00079=166821,969292,1072076
BC00080=166821,969292,1072076
BC00081=166821,969292,1072076
BC00082=166820,969293,1072075
BC00083=274128,961901,1072075
BC00084=274128,961901,1072075
BC00085=274128,961901,1072075
BC00086=274128,961901,1072075
BC00087=274128,961901,1072075
BC00088=274128,961901,1072075
BC00089=274128,961901,1072075
BC00090=274128,961901,1072075
BC00091=274128,961901,1072071
BC00092=274128,961901,1072071
BC00093=274128,961901,1072071
BC00094=274128,961901,1072071
BC00095=274128,961901,1072071
BC00096=274128,961901,1072071
BC00097=253787,895567,1072071
BC00098=253787,895567,1066387
BC00099=253787,895567,1066387
BC00100=253787,895567,1066387
BC00101=253787,895567,1066387
BC00102=253787,895567,1066387
BC00103=253787,895567,1066387
BC00104=253787,895567,1066387
BC00105=332690,882659,1072071
BC00106=352776,943841,1062049
BC00107=352776,943841,1056120
BC00108=352776,943841,1056120
BC00109=352776,943841,1056120
BC00110=352776,943841,1056120
BC00111=352776,943841,1056120
BC00112=352776,943841,1056120
BC00113=352776,943841,1056120
BC00114=352776,943841,1056120
BC00115=352776,943841,1056120
BC00116=352776,943841,1056120
BC00117=352776,943841,1056120
BC00118=352776,943841,1056120
BC00119=352776,943841,1056120
BC00120=310169,911968,1073469
BC00121=291623,911782,1074972
BC00122=268902,904998,1073205
BC00123=268902,904998,1073205
BC00124=268902,904998,1073205
BC00125=268902,904998,1073205
BC00126=268902,904998,1073205
BC00127=268902,904998,1073205
BC00128=320878,904998,1073205
BC00129=320878,904998,1073205
BC00130=320878,904998,1073205
BC00131=320878,904998,1073205
BC00132=320878,904998,1073205
BC00133=320878,904998,1073205
BC00134=320878,904998,1073205
BC00135=213337,904998,1073205
BC00136=213337,904998,1068795
BC00137=213337,904998,1068795
BC00138=213337,904998,1068795
BC00139=213337,904998,1068795
BC00140=213337,904998,1068795
BC00141=213337,904998,1068795
BC00142=170757,904998,1068795
BC00143=170757,904998,1068795
BC00144=170757,904998,1068795
BC00145=170757,904998,1068795
BC00146=170757,904998,1068795
BC00147=170757,904998,1068795
BC00148=193221,1067506,1068795
BC00149=193221,1067506,1068795
BC00150=193221,1067506,1068795
BC00151=193221,1067506,1068795
BC00152=193221,1067506,1068795
BC00153=193221,1067506,1068795
BC00154=193221,1067506,1068795
BC00155=199711,1067506,1068794
BC00156=207788,1067506,1068792
BC00157=207788,1067506,1068790
BC00158=207788,1067506,1068792
BC00159=207788,1067506,1068792
BC00160=207788,1067506,1068792
BC00161=207788,1067506,1073587
BC00162=282406,880495,1068555
BC00163=282406,880495,1066387
BC00164=282404,880494,1066387
BC00165=282404,880494,1066387
BC00166=282404,880494,1066387
BC00167=282404,880494,1066387
BC00168=282404,880494,1066387
BC00169=100678,973416,1072339
BC00170=113353,1001451,1072339
BC00171=107557,1002422,1072440
BC00172=36539,1014323,1073683
BC00173=30635,1015327,1073683
BC00174=112239,958761,1072440
BC00175=388770,864829,1072440
BC00176=395574,924315,1072438
BC00177=396601,933289,1072438
BC00178=396601,933289,1072438
BC00179=396601,933289,1072438
BC00180=396601,933289,1072438
BC00181=316599,920939,1070848
BC00182=213337,904998,1068795
BC00183=213337,904998,1068795
BC00184=213337,904998,1068795
BC00185=213337,904998,1068795
BC00186=213337,904998,1068795
BC00187=213337,904998,1068795
BC00188=327385,904998,1068795
BC00189=316881,884304,1068795
BC00190=316881,884304,1068795
BC00191=316881,884304,1068795
BC00192=316881,884304,1068795
BC00193=316881,884304,1068795
BC00194=316098,887435,1068795
BC00195=274128,953808,1072075
BC00196=274128,961901,1072075
BC00197=274129,961901,1072073
BC00198=274129,961901,1072073
BC00199=274129,961901,1072073
BC00200=274129,961901,1072073
BC00201=274129,961901,1072073
BC00202=191184,974268,1072073
BC00203=191184,974268,1072073
BC00204=191184,974268,1072073
BC00205=191184,974268,1072073
BC00206=191184,974268,1072073
BC00207=191184,974268,1072073
BC00208=191184,974268,1072073
BC00209=181213,974268,1072073
BC00210=181213,974268,1072073
BC00211=181213,974268,1072073
BC00212=102087,963066,1072073
BC00213=102087,963066,1072073
BC00214=102087,963066,1072073
BC00215=102087,963066,1072073
BC00216=102087,963066,1072073
BC00217=102087,963066,1072070
BC00218=124233,740604,1070750
BC00219=168854,844547,1075175
BC00220=168854,844547,1075175
BC00221=168854,844547,1075175
BC00222=168854,844547,1075175
BC00223=168854,844547,1075175
BC00224=168854,844547,1075175
BC00225=168854,844547,1075175
BC00226=168854,844547,1075175
BC00227=168854,844547,1075175
BC00228=168854,844547,1075175
BC00229=125556,866811,1075175
BC00230=125556,866811,1075175
BC00231=125556,866811,1075175
BC00232=125556,866811,1075175
BC00233=125556,866811,1075175
BC00234=125556,866811,1075175
BC00235=125556,866811,1075175
BC00236=125556,866811,1075175
BC00237=125556,866811,1075175
BC00238=125556,866811,1075175
BC00239=94030,883389,1075175
BC00240=94030,883389,1075175
BC00241=94030,883389,1075175
BC00242=94030,883389,1075175
BC00243=94030,883389,1075175
BC00244=94030,883389,1075175
BC00245=94030,883389,1075175
BC00246=94030,883389,1075175
BC00247=94030,883389,1075175
BC00248=94030,883389,1075175
BC00249=94030,883389,1075175
BC00250=254016,900546,1075175
BC00251=254016,900546,1075175
BC00252=254016,900546,1075175
BC00253=254016,900546,1075175
BC00254=254016,900546,1075175
BC00255=254016,900546,1075175
BC00256=254016,900546,1075175
BC00257=254016,900546,1075175
BC00258=254016,900546,1075175
BC00259=254016,900546,1075175
BC00260=254016,900546,1075175
BC00261=131751,862217,1075175
BC00262=131751,862217,1075175
BC00263=131751,862217,1075175
BC00264=131751,862217,1075175
BC00265=131751,862217,1075175
BC00266=131751,862217,1075175
BC00267=131751,862217,1075175
BC00268=131751,862217,1075175
BC00269=131751,862217,1075175
BC00270=131751,862217,1075175
BC00271=107480,867622,1075175
BC00272=36182,883500,1075175
BC00273=36182,883500,1075175
BC00274=36182,883500,1075175
BC00275=36182,883500,1075175
BC00276=36182,883500,1075175
BC00277=36182,883500,1075175
BC00278=36182,883500,1075175
BC00279=36182,883500,1075175
BC00280=36182,883500,1075175
BC00281=36182,883500,1075175
BC00282=65366,862824,1075175
BC00283=79958,852485,1075175
BC00284=79958,852485,1075175
BC00285=79958,852485,1075175
BC00286=79958,852485,1075175
BC00287=79958,852485,1075175
BC00288=79958,852485,1075175
BC00289=79958,852485,1075175
BC00290=79958,852485,1075175
BC00291=79958,852485,1075175
BC00292=79958,852485,1075175
BC00293=79958,852485,1075175
BC00294=79958,852485,1075175
BC00295=79958,852485,1075175
BC00296=253095,795778,1075175
BC00297=253095,795778,1075175
BC00298=253095,795778,1075175
BC00299=253095,795778,1075175
BC00300=253095,795778,1075175
BC00301=253095,795778,1075175
BC00302=253095,795778,1075175
BC00303=253095,795778,1075175
BC00304=253095,795778,1075175
BC00305=253095,795778,1075175
BC00306=253095,795778,1075175
BC00307=277970,773099,1075175
BC00308=277970,773099,1075175
BC00309=277970,773099,1075175
BC00310=277970,773099,1075175
BC00311=277970,773099,1075175
BC00312=277970,773099,1075175
BC00313=277970,773099,1075175
BC00314=277970,773099,1075175
BC00315=277970,773099,1075175
BC00316=277970,773099,1075175
BC00317=277970,773099,1075175
BC00318=277970,773099,1075175
BC00319=391401,773564,1075175
BC00320=391401,773564,1075175
BC00321=391401,773564,1075175
BC00322=391401,773564,1075175
BC00323=391401,773564,1075175
BC00324=391401,773564,1075175
BC00325=391401,773564,1075175
BC00326=391401,773564,1075175
BC00327=391401,773564,1075175
BC00328=391401,773564,1075175
BC00329=391279,862949,1075175
BC00330=391279,862949,1075175
BC00331=391279,862949,1075175
BC00332=391279,862949,1075175
BC00333=391279,862949,1075175
BC00334=391279,862949,1075175
BC00335=391279,862949,1075175
BC00336=391279,862949,1075175
BC00337=391279,862949,1075175
BC00338=391279,862949,1075175
BC00339=391279,862949,1075175
BC00340=356671,865533,1075175
BC00341=337474,866966,1075175
BC00342=275808,871571,1075175
BC00343=275808,871571,1075175
BC00344=275808,871571,1075175
BC00345=275808,871571,1075175
BC00346=275808,871571,1075175
BC00347=275808,871571,1075175
BC00348=275808,871571,1075175
BC00349=275808,871571,1075175
BC00350=275808,871571,1075175
BC00351=275808,871571,1075175
BC00352=275808,871571,1075175
BC00353=307223,910718,1075175
BC00354=307223,910718,1075175
BC00355=307223,910718,1075175
BC00356=307223,910718,1075175
BC00357=307223,910718,1075175
BC00358=307223,910718,1075175
BC00359=307223,910718,1075175
BC00360=307223,910718,1075175
BC00361=307223,910718,1075175
BC00362=307223,910718,1075175
BC00363=285896,934777,1075175
BC00364=287314,930132,1075175
BC00365=287881,928273,1075169
BC00366=287881,928274,1075175
BC00367=287881,928274,1075175
BC00368=331662,908320,1075175
BC00369=298889,925540,1075175
BC00370=304335,922407,1075175
BC00371=306243,923246,1075175
BC00372=311013,925342,1075175
BC00373=310992,925340,1075175
BC00374=288951,837561,1075175
BC00375=272420,771727,1075175
BC00376=272441,771729,1075175
BC00377=274912,778521,1075175
BC00378=275901,781238,1075175
BC00379=275901,781238,1075175
BC00380=275901,781238,1075175
BC00381=271752,783389,1075175
BC00382=238445,800873,1075175
BC00383=234327,803060,1075175
BC00384=233339,800343,1075175
BC00385=230868,793551,1075175
BC00386=78008,861005,1075175
BC00387=77769,868446,1075175
BC00388=77674,871423,1075175
BC00389=77674,871423,1075175
BC00390=77674,871423,1075175
BC00391=23886,880099,1075175
BC00392=19182,880858,1075175
BC00393=19277,877881,1075175
BC00394=19516,870440,1075175
BC00395=19495,870438,1075175
BC00396=326092,855697,1075175
BC00397=326092,855697,1075175
BC00398=398174,852232,1075175
BC00399=398174,857485,1075175
BC00400=398174,859586,1075175
BC00401=398174,859586,1075175
BC00402=398174,859586,1075175
BC00403=371813,869160,1075175
BC00404=367110,869924,1075175
BC00405=367173,867823,1075175
BC00406=367173,867823,1075175
BC00407=367173,867823,1075175
BC00408=360387,856598,1075175
BC00409=311250,775314,1075175
BC00410=310674,772108,1075175
BC00411=310157,770863,1075175
BC00412=310443,770826,1075175
BC00413=310443,770826,1075175
BC00414=310157,770863,1075175
BC00415=281252,771527,1075175
BC00416=281201,772763,1075175
BC00417=283941,775788,1075175
BC00418=283920,775786,1075175
BC00419=277373,824158,1075175
BC00420=275378,838906,1075175
BC00421=277972,845384,1075175
BC00422=279902,846207,1075175
BC00423=279010,847975,1075175
BC00424=279010,847975,1075175
BC00425=308125,844091,1075175
BC00426=270491,850162,1075175
BC00427=273128,849737,1075175
BC00428=273830,846973,1075175
BC00429=275584,840064,1075175
BC00430=275563,840061,1075175
BC00431=324608,813796,1075175
BC00432=398174,774398,1075175
BC00433=398174,774401,1075175
BC00434=398174,771767,1075175
BC00435=398174,771517,1075173
BC00436=398174,770713,1075175
BC00437=398174,770713,1075175
BC00438=345888,773938,1075175
BC00439=391446,773901,1075175
BC00440=395311,773894,1075175
BC00441=395311,773894,1075175
BC00442=395554,778391,1075175
BC00443=395533,778388,1075175
BC00444=244947,801075,1075175
BC00445=66752,827920,1075175
BC00446=66773,827923,1075175
BC00447=63808,834893,1075175
BC00448=62622,837682,1075175
BC00449=62622,837682,1075175
BC00450=62622,837682,1075175
BC00451=65024,838688,1075175
BC00452=67719,839810,1075175
BC00453=67719,839810,1075175
BC00454=71870,830051,1075175
BC00455=97426,846419,1075175
BC00456=97270,849222,1075175
BC00457=97270,849222,1075175
BC00458=97270,849222,1075175
BC00459=92568,849992,1075175
BC00460=61997,854937,1075175
BC00461=64634,854514,1075175
BC00462=65336,851751,1075175
BC00463=84699,851770,1075175
BC00464=124914,851811,1075175
BC00465=124935,851814,1075175
BC00466=122737,858395,1075175
BC00467=121858,861028,1075175
BC00468=121858,861028,1075175
BC00469=121858,861028,1075175
BC00470=124620,862466,1075175
BC00471=125499,859833,1075175
BC00472=127697,853251,1075175
BC00473=127676,853249,1075175
BC00474=204722,814942,1075175
BC00475=204743,814944,1075175
BC00476=206674,821646,1075175
BC00477=207446,824327,1075175
BC00478=207446,824327,1075175
BC00479=207446,824327,1075175
BC00480=204611,825752,1075175
BC00481=203320,826401,1075175
BC00482=200485,827827,1075175
BC00483=199712,825146,1075175
BC00484=197782,818445,1075175
BC00485=159365,837791,1075175
BC00486=161435,844430,1075175
BC00487=162263,847086,1075175
BC00488=162263,847086,1075175
BC00489=162263,847086,1075175
BC00490=158269,849138,1075175
BC00491=157441,846482,1075175
BC00492=155371,839843,1075175
BC00493=121548,857305,1075175
BC00494=123718,863898,1075175
BC00495=124587,866535,1075175
BC00496=124587,866535,1075175
BC00497=124587,866535,1075175
BC00498=120591,868620,1075175
BC00499=119723,865983,1075175
BC00500=117552,859390,1075175
BC00501=117531,859387,1075175
BC00502=246992,896371,1075175
BC00503=220074,877634,1075175
BC00504=181712,850933,1075175
BC00505=181712,850933,1075175
BC00506=238846,900446,1075175
BC00507=238846,900446,1075175
BC00508=233667,887804,1075175
BC00509=233736,914980,1075175
BC00510=230071,889541,1075175
BC00511=233789,896183,1075175
BC00512=229861,888764,1075175
BC00513=221340,873628,1075175
BC00514=204000,858703,1075175
BC00515=181712,850933,1075175
BC00516=163054,850862,1075175
BC00517=145387,858647,1075175
BC00518=143913,859593,1075175
BC00519=142936,860330,1075175
BC00520=147400,860834,1075175
BC00521=147400,860834,1075175
BC00522=147400,860834,1075175
BC00523=147209,858034,1075175
BC00524=146826,852434,1075175
BC00525=162823,738758,1075175
BC00526=162823,738758,1075175
BC00527=162823,738758,1075175
BC00528=162469,668315,1065860
BC00529=132836,722637,395133
BC00530=132836,785697,289538
BC00531=120112,840943,355403
BC00532=120112,840943,355403
BC00533=120112,840943,355403
BC00534=120112,840943,355403
BC00535=120112,840943,355403
BC00536=120112,840943,355403
BC00537=120112,840943,355403
BC00538=120112,840943,355403
BC00539=120112,840943,355403
BC00540=120112,840943,355403
BC00541=112990,845108,322924
BC00542=112990,845108,322924
BC00543=112990,845108,322924
BC00544=112990,845108,322924
BC00545=112990,845108,322924
BC00546=112990,845108,322924
BC00547=112990,845108,322924
BC00548=112990,845108,322924
BC00549=104813,823501,393324
BC00550=104813,823501,393324
BC00551=104813,760081,393324
BC00552=248254,760081,393324
BC00553=248246,711751,217199
BC00554=248240,678922,53
BC00555=292488,813118,262788
BC00556=292488,813118,262788
BC00557=292487,813119,262787
BC00558=292488,813118,262788
BC00559=292488,813118,262788
BC00560=292487,813119,262787
BC00561=292487,813119,262787
BC00562=292487,813119,262787
BC00563=292487,813119,262787
BC00564=292487,813119,262787
BC00565=292488,813118,262788
BC00566=292488,813118,262788
BC00567=292488,813118,262788
BC00568=274061,782472,233150
BC00569=216295,686398,140238
BC00570=267150,771347,84751
BC00571=267150,771347,84751
BC00572=267150,771347,84751
BC00573=267149,771347,84748
BC00574=267150,771347,84751
BC00575=267150,771347,84751
BC00576=267149,771347,84748
BC00577=267149,771347,84748
BC00578=267149,771347,84748
BC00579=267149,771347,84748
BC00580=267149,771347,84748
BC00581=267149,771347,84748
BC00582=267150,771347,84751
BC00583=267150,771347,84751
BC00584=248348,722947,225922
BC00585=227130,668325,385240
BC00586=89228,669140,483629
BC00587=85891,769521,393324
BC00588=85891,823501,393324
BC00589=78694,819217,285317
BC00590=80911,824247,266429
BC00591=81798,826258,258874
BC00592=81798,826258,258874
BC00593=81798,826258,258874
BC00594=77667,828574,258907
BC00595=73118,831123,258944
BC00596=68987,833438,258977
BC00597=68100,831426,266531
BC00598=65882,826396,285419
BC00599=89795,837211,285494
BC00600=92010,842241,266606
BC00601=92896,844254,259052
BC00602=92896,844254,259052
BC00603=92896,844254,259052
BC00604=92896,844254,259052
BC00605=92896,844254,259052
BC00606=92896,844254,259052
BC00607=85891,823501,393324
BC00608=85891,764660,393324
BC00609=85891,709426,393324
BC00610=162291,708666,208254
BC00611=248240,707811,53
BC00612=248240,740511,53
BC00613=263228,763657,33242
BC00614=270136,774326,48540
BC00615=270136,774326,48540
BC00616=289480,804199,91375
BC00617=289480,804199,91375
BC00618=270136,774326,48540
BC00619=270136,774326,48540
BC00620=270419,774762,49166
BC00621=268962,774570,99865
BC00622=269143,774832,97699
BC00623=269143,774832,97699
BC00624=271008,780091,86007
BC00625=271008,780091,86007
BC00626=269143,774832,97699
BC00627=269143,774832,97699
BC00628=268098,775090,99700
BC00629=248240,678922,53
BC00630=248240,678922,53
BC00631=325149,799380,131072
BC00632=325149,799380,131072
BC00633=325149,799379,131071
BC00634=325149,799380,131072
BC00635=325149,799380,131072
BC00636=325149,799379,131071
BC00637=325149,799379,131071
BC00638=325149,799379,131071
BC00639=325149,799379,131071
BC00640=325149,799379,131071
BC00641=325149,799379,131071
BC00642=325149,799380,131072
BC00643=309454,697955,17856
BC00644=284186,811897,242158
BC00645=284186,811897,242158
BC00646=284186,811897,242158
BC00647=284186,811897,242158
BC00648=284186,811897,242158
BC00649=284186,811897,242158
BC00650=284186,811897,242158
BC00651=284186,811897,242158
BC00652=294965,806037,143387
BC00653=294965,806037,143387
BC00654=294965,806037,143387
BC00655=294965,806037,143387
BC00656=294965,806037,143387
BC00657=294965,806037,143387
BC00658=294965,806037,143387
BC00659=294965,806037,143387
BC00660=294965,806037,143387
BC00661=346884,805648,147012
BC00662=344714,817518,131657
BC00663=344714,817518,131657
BC00664=344714,817518,131657
BC00665=344714,817518,131657
BC00666=344714,817518,131657
BC00667=344714,817518,131657
BC00668=344714,817518,131657
BC00669=344714,817518,131657
BC00670=344714,817518,131657
BC00671=344714,817518,131657
BC00672=344714,817518,131657
BC00673=344714,668458,131654
BC00674=142431,668458,131654
EC00000=798156,1112951
EC00001=798156,1112951
EC00002=798156,1112951
EC00003=798156,1112951
EC00004=798156,1112951
EC00005=798156,1112951
EC00006=798156,1112951
EC00007=798156,1112951
EC00008=798156,1112951
EC00009=798156,1112951
EC00010=798156,1112951
EC00011=798156,1112951
EC00012=798156,1112951
EC00013=798156,1112951
EC00014=798156,1112951
EC00015=798156,1112951
EC00016=798156,1112951
EC00017=798156,1112951
EC00018=798156,1112951
EC00019=798156,1112951
EC00020=798156,1112951
EC00021=798156,1112951
EC00022=798156,1112951
EC00023=798156,1112951
EC00024=798156,1112951
EC00025=798156,1112951
EC00026=798156,1112951
EC00027=798156,1112951
EC00028=798156,1112951
EC00029=798156,1112951
EC00030=798156,1112951
EC00031=798156,1112951
EC00032=798156,1112951
EC00033=798156,1112951
EC00034=798156,1112951
EC00035=798156,1112951
EC00036=798156,1112951
EC00037=798156,1112951
EC00038=798156,1112951
EC00039=798156,1112951
EC00040=798156,1112951
EC00041=798156,1112951
EC00042=798156,1112951
EC00043=798156,1112951
EC00044=798156,1112951
EC00045=798156,1112951
EC00046=798156,1112951
EC00047=798156,1112951
EC00048=798156,1112951
EC00049=798155,1112950
EC00050=798155,1112950
EC00051=798155,1112950
EC00052=798155,1112950
EC00053=798155,1112950
EC00054=798155,1112950
EC00055=798155,1112950
EC00056=798155,1112950
EC00057=798155,1112950
EC00058=798155,1112950
EC00059=798155,1112950
EC00060=798155,1112950
EC00061=798155,1112950
EC00062=798155,1112950
EC00063=798155,1112950
EC00064=798155,1112950
EC00065=798155,1112950
EC00066=798155,1112950
EC00067=798154,1112950
EC00068=798155,1112950
EC00069=798155,1112950
EC00070=798155,1112950
EC00071=798155,1112950
EC00072=798155,1112950
EC00073=798155,1112950
EC00074=798155,1112950
EC00075=798155,1112950
EC00076=798155,1112950
EC00077=798155,1112950
EC00078=798155,1112950
EC00079=798155,1112950
EC00080=798155,1112950
EC00081=798155,1112950
EC00082=798154,1112949
EC00083=798154,1112949
EC00084=798154,1112949
EC00085=798154,1112949
EC00086=798154,1112949
EC00087=798154,1112949
EC00088=798154,1112949
EC00089=798154,1112949
EC00090=798154,1112949
EC00091=798153,1112947
EC00092=798153,1112947
EC00093=798153,1112947
EC00094=798153,1112947
EC00095=798153,1112947
EC00096=798153,1112947
EC00097=798153,1112947
EC00098=798153,1112947
EC00099=798153,1112947
EC00100=798153,1112947
EC00101=798153,1112947
EC00102=798153,1112947
EC00103=798153,1112947
EC00104=798153,1112947
EC00105=798153,1112947
EC00106=798153,1112947
EC00107=798153,1112947
EC00108=798153,1112947
EC00109=798153,1112947
EC00110=798153,1112947
EC00111=798153,1112947
EC00112=798153,1112947
EC00113=798153,1112947
EC00114=798153,1112947
EC00115=798153,1112947
EC00116=798153,1112947
EC00117=798153,1112947
EC00118=798153,1112947
EC00119=798153,1112947
EC00120=798153,1112947
EC00121=798153,1112947
EC00122=798152,1112946
EC00123=798152,1112946
EC00124=798152,1112946
EC00125=798152,1112946
EC00126=798152,1112946
EC00127=798152,1112946
EC00128=798152,1112946
EC00129=798152,1112946
EC00130=798152,1112946
EC00131=798152,1112946
EC00132=798152,1112946
EC00133=798152,1112946
EC00134=798152,1112946
EC00135=798152,1112946
EC00136=798152,1112946
EC00137=798152,1112946
EC00138=798152,1112946
EC00139=798152,1112946
EC00140=798152,1112946
EC00141=798152,1112946
EC00142=798152,1112946
EC00143=798152,1112946
EC00144=798152,1112946
EC00145=798152,1112946
EC00146=798152,1112946
EC00147=798152,1112946
EC00148=798152,1112946
EC00149=798152,1112946
EC00150=798152,1112946
EC00151=798152,1112946
EC00152=798152,1112946
EC00153=798152,1112946
EC00154=798152,1112946
EC00155=798151,1112945
EC00156=798149,1112944
EC00157=798148,1112944
EC00158=798149,1112944
EC00159=798149,1112944
EC00160=798149,1112944
EC00161=798149,1112944
EC00162=798153,1112947
EC00163=798153,1112947
EC00164=798152,1112946
EC00165=798152,1112946
EC00166=798152,1112946
EC00167=798152,1112946
EC00168=798152,1112946
EC00169=798152,1112946
EC00170=798152,1112946
EC00171=798152,1112946
EC00172=798152,1112946
EC00173=798152,1112946
EC00174=798152,1112946
EC00175=798152,1112946
EC00176=798151,1112945
EC00177=798151,1112945
EC00178=798151,1112945
EC00179=798151,1112945
EC00180=798151,1112945
EC00181=798151,1112945
EC00182=798152,1112946
EC00183=798152,1112946
EC00184=798152,1112946
EC00185=798152,1112946
EC00186=798152,1112946
EC00187=798152,1112946
EC00188=798152,1112946
EC00189=798152,1112946
EC00190=798152,1112946
EC00191=798152,1112946
EC00192=798152,1112946
EC00193=798152,1112946
EC00194=798152,1112946
EC00195=798154,1112949
EC00196=798154,1112949
EC00197=798153,1112947
EC00198=798153,1112947
EC00199=798153,1112947
EC00200=798153,1112947
EC00201=798153,1112947
EC00202=798153,1112947
EC00203=798153,1112947
EC00204=798153,1112947
EC00205=798153,1112947
EC00206=798153,1112947
EC00207=798153,1112947
EC00208=798153,1112947
EC00209=798153,1112947
EC00210=798153,1112947
EC00211=798153,1112947
EC00212=798153,1112947
EC00213=798153,1112947
EC00214=798153,1112947
EC00215=798153,1112947
EC00216=798153,1112947
EC00217=798152,1112946
EC00218=798152,1112946
EC00219=975524,1112951
EC00220=975524,1112951
EC00221=975524,1112951
EC00222=975524,1112951
EC00223=975524,1112951
EC00224=975524,1112951
EC00225=975524,1112951
EC00226=975524,1112951
EC00227=975524,1112951
EC00228=975524,1112951
EC00229=975524,1112951
EC00230=975524,1112951
EC00231=975524,1112951
EC00232=975524,1112951
EC00233=975524,1112951
EC00234=975524,1112951
EC00235=975524,1112951
EC00236=975524,1112951
EC00237=975524,1112951
EC00238=975524,1112951
EC00239=975524,1112951
EC00240=975524,1112951
EC00241=975524,1112951
EC00242=975524,1112951
EC00243=975524,1112951
EC00244=975524,1112951
EC00245=975524,1112951
EC00246=975524,1112951
EC00247=975524,1112951
EC00248=975524,1112951
EC00249=975524,1112951
EC00250=975524,1112951
EC00251=975524,1112951
EC00252=975524,1112951
EC00253=975524,1112951
EC00254=975524,1112951
EC00255=975524,1112951
EC00256=975524,1112951
EC00257=975524,1112951
EC00258=975524,1112951
EC00259=975524,1112951
EC00260=975524,1112951
EC00261=975524,1112951
EC00262=975524,1112951
EC00263=975524,1112951
EC00264=975524,1112951
EC00265=975524,1112951
EC00266=975524,1112951
EC00267=975524,1112951
EC00268=975524,1112951
EC00269=975524,1112951
EC00270=975524,1112951
EC00271=975524,1112951
EC00272=975524,1112951
EC00273=975524,1112951
EC00274=975524,1112951
EC00275=975524,1112951
EC00276=975524,1112951
EC00277=975524,1112951
EC00278=975524,1112951
EC00279=975524,1112951
EC00280=975524,1112951
EC00281=975524,1112951
EC00282=975524,1112951
EC00283=975524,1112951
EC00284=975524,1112951
EC00285=975524,1112951
EC00286=975524,1112951
EC00287=975524,1112951
EC00288=975524,1112951
EC00289=975524,1112951
EC00290=975524,1112951
EC00291=975524,1112951
EC00292=975524,1112951
EC00293=975524,1112951
EC00294=975524,1112951
EC00295=975524,1112951
EC00296=975524,1112951
EC00297=975524,1112951
EC00298=975524,1112951
EC00299=975524,1112951
EC00300=975524,1112951
EC00301=975524,1112951
EC00302=975524,1112951
EC00303=975524,1112951
EC00304=975524,1112951
EC00305=975524,1112951
EC00306=975524,1112951
EC00307=975524,1112951
EC00308=975524,1112951
EC00309=975524,1112951
EC00310=975524,1112951
EC00311=975524,1112951
EC00312=975524,1112951
EC00313=975524,1112951
EC00314=975524,1112951
EC00315=975524,1112951
EC00316=975524,1112951
EC00317=975524,1112951
EC00318=975524,1112951
EC00319=975524,1112951
EC00320=975524,1112951
EC00321=975524,1112951
EC00322=975524,1112951
EC00323=975524,1112951
EC00324=975524,1112951
EC00325=975524,1112951
EC00326=975524,1112951
EC00327=975524,1112951
EC00328=975524,1112951
EC00329=975524,1112951
EC00330=975524,1112951
EC00331=975524,1112951
EC00332=975524,1112951
EC00333=975524,1112951
EC00334=975524,1112951
EC00335=975524,1112951
EC00336=975524,1112951
EC00337=975524,1112951
EC00338=975524,1112951
EC00339=975524,1112951
EC00340=975524,1112951
EC00341=975524,1112951
EC00342=975524,1112951
EC00343=975524,1112951
EC00344=975524,1112951
EC00345=975524,1112951
EC00346=975524,1112951
EC00347=975524,1112951
EC00348=975524,1112951
EC00349=975524,1112951
EC00350=975524,1112951
EC00351=975524,1112951
EC00352=975524,1112951
EC00353=975524,1112951
EC00354=975524,1112951
EC00355=975524,1112951
EC00356=975524,1112951
EC00357=975524,1112951
EC00358=975524,1112951
EC00359=975524,1112951
EC00360=975524,1112951
EC00361=975524,1112951
EC00362=975524,1112951
EC00363=975524,1112951
EC00364=975524,1112951
EC00365=975518,1112948
EC00366=975524,1112951
EC00367=975524,1112951
EC00368=975524,1112951
EC00369=975524,1112951
EC00370=975524,1112951
EC00371=975524,1112951
EC00372=975524,1112951
EC00373=975524,1112951
EC00374=975524,1112951
EC00375=975524,1112951
EC00376=975524,1112951
EC00377=975524,1112951
EC00378=975524,1112951
EC00379=975524,1112951
EC00380=975524,1112951
EC00381=975524,1112951
EC00382=975524,1112951
EC00383=975524,1112951
EC00384=975524,1112951
EC00385=975524,1112951
EC00386=975524,1112951
EC00387=975524,1112951
EC00388=975524,1112951
EC00389=975524,1112951
EC00390=975524,1112951
EC00391=975524,1112951
EC00392=975524,1112951
EC00393=975524,1112951
EC00394=975524,1112951
EC00395=975524,1112951
EC00396=975524,1112951
EC00397=975524,1112951
EC00398=975524,1112951
EC00399=975524,1112951
EC00400=975524,1112951
EC00401=975524,1112951
EC00402=975524,1112951
EC00403=975524,1112951
EC00404=975524,1112951
EC00405=975524,1112951
EC00406=975524,1112951
EC00407=975524,1112951
EC00408=975524,1112951
EC00409=975524,1112951
EC00410=975524,1112951
EC00411=975524,1112951
EC00412=975524,1112951
EC00413=975524,1112951
EC00414=975524,1112951
EC00415=975524,1112951
EC00416=975524,1112951
EC00417=975524,1112951
EC00418=975524,1112951
EC00419=975524,1112951
EC00420=975524,1112951
EC00421=975524,1112951
EC00422=975524,1112951
EC00423=975524,1112951
EC00424=975524,1112951
EC00425=975524,1112951
EC00426=975524,1112951
EC00427=975524,1112951
EC00428=975524,1112951
EC00429=975524,1112951
EC00430=975524,1112951
EC00431=975524,1112951
EC00432=975524,1112951
EC00433=975524,1112951
EC00434=975524,1112951
EC00435=975522,1112950
EC00436=975524,1112951
EC00437=975524,1112951
EC00438=975524,1112951
EC00439=975524,1112951
EC00440=975524,1112951
EC00441=975524,1112951
EC00442=975524,1112951
EC00443=975524,1112951
EC00444=975524,1112951
EC00445=975524,1112951
EC00446=975524,1112951
EC00447=975524,1112951
EC00448=975524,1112951
EC00449=975524,1112951
EC00450=975524,1112951
EC00451=975524,1112951
EC00452=975524,1112951
EC00453=975524,1112951
EC00454=975524,1112951
EC00455=975524,1112951
EC00456=975524,1112951
EC00457=975524,1112951
EC00458=975524,1112951
EC00459=975524,1112951
EC00460=975524,1112951
EC00461=975524,1112951
EC00462=975524,1112951
EC00463=975524,1112951
EC00464=975524,1112951
EC00465=975524,1112951
EC00466=975524,1112951
EC00467=975524,1112951
EC00468=975524,1112951
EC00469=975524,1112951
EC00470=975524,1112951
EC00471=975524,1112951
EC00472=975524,1112951
EC00473=975524,1112951
EC00474=975524,1112951
EC00475=975524,1112951
EC00476=975524,1112951
EC00477=975524,1112951
EC00478=975524,1112951
EC00479=975524,1112951
EC00480=975524,1112951
EC00481=975524,1112951
EC00482=975524,1112951
EC00483=975524,1112951
EC00484=975524,1112951
EC00485=975524,1112951
EC00486=975524,1112951
EC00487=975524,1112951
EC00488=975524,1112951
EC00489=975524,1112951
EC00490=975524,1112951
EC00491=975524,1112951
EC00492=975524,1112951
EC00493=975524,1112951
EC00494=975524,1112951
EC00495=975524,1112951
EC00496=975524,1112951
EC00497=975524,1112951
EC00498=975524,1112951
EC00499=975524,1112951
EC00500=975524,1112951
EC00501=975524,1112951
EC00502=975524,1112951
EC00503=975524,1112951
EC00504=975524,1112951
EC00505=975524,1112951
EC00506=975524,1112951
EC00507=975524,1112951
EC00508=975524,1112951
EC00509=975524,1112951
EC00510=975524,1112951
EC00511=975524,1112951
EC00512=975524,1112951
EC00513=975524,1112951
EC00514=975524,1112951
EC00515=975524,1112951
EC00516=975524,1112951
EC00517=975524,1112951
EC00518=975524,1112951
EC00519=975524,1112951
EC00520=975524,1112951
EC00521=975524,1112951
EC00522=975524,1112951
EC00523=975524,1112951
EC00524=975524,1112951
EC00525=975524,1112951
EC00526=798156,1112951
EC00527=798156,1112951
EC00528=798154,1112951
EC00529=798156,1112951
EC00530=798156,1112951
EC00531=798156,1112951
EC00532=798156,1112951
EC00533=798156,1112951
EC00534=798156,1112951
EC00535=798156,1112951
EC00536=798156,1112951
EC00537=798156,1112951
EC00538=798156,1112951
EC00539=798156,1112951
EC00540=798156,1112951
EC00541=798156,1112951
EC00542=798156,1112951
EC00543=798156,1112951
EC00544=798156,1112951
EC00545=798156,1112951
EC00546=798156,1112951
EC00547=798156,1112951
EC00548=798156,1112951
EC00549=798156,1112951
EC00550=798156,1112951
EC00551=798156,1112951
EC00552=798156,1112951
EC00553=798156,1112951
EC00554=798156,1112951
EC00555=798156,1112951
EC00556=798156,1112951
EC00557=798155,1112950
EC00558=798156,1112951
EC00559=798156,1112951
EC00560=798155,1112950
EC00561=798155,1112950
EC00562=798155,1112950
EC00563=798155,1112950
EC00564=798155,1112950
EC00565=798156,1112951
EC00566=798156,1112951
EC00567=798156,1112951
EC00568=798156,1112951
EC00569=798156,1112951
EC00570=798156,1112951
EC00571=798156,1112951
EC00572=798156,1112951
EC00573=798155,1112949
EC00574=798156,1112951
EC00575=798156,1112951
EC00576=798155,1112949
EC00577=798155,1112949
EC00578=798155,1112949
EC00579=798155,1112949
EC00580=798155,1112949
EC00581=798155,1112949
EC00582=798156,1112951
EC00583=798156,1112951
EC00584=798156,1112951
EC00585=798156,1112951
EC00586=798156,1112951
EC00587=798156,1112951
EC00588=798156,1112951
EC00589=798156,1112951
EC00590=798156,1112951
EC00591=798156,1112951
EC00592=798156,1112951
EC00593=798156,1112951
EC00594=798156,1112951
EC00595=798156,1112951
EC00596=798156,1112951
EC00597=798156,1112951
EC00598=798156,1112951
EC00599=798156,1112951
EC00600=798156,1112951
EC00601=798156,1112951
EC00602=798156,1112951
EC00603=798156,1112951
EC00604=798156,1112951
EC00605=798156,1112951
EC00606=798156,1112951
EC00607=798156,1112951
EC00608=798156,1112951
EC00609=798156,1112951
EC00610=798156,1112951
EC00611=798156,1112951
EC00612=798156,1112951
EC00613=798156,1112951
EC00614=798155,1112950
EC00615=798155,1112950
EC00616=798156,1112951
EC00617=798156,1112951
EC00618=798155,1112950
EC00619=798155,1112950
EC00620=798155,1112950
EC00621=798155,1112950
EC00622=798155,1112950
EC00623=798155,1112950
EC00624=798156,1112951
EC00625=798156,1112951
EC00626=798155,1112950
EC00627=798155,1112950
EC00628=798155,1112950
EC00629=798156,1112951
EC00630=798156,1112951
EC00631=798156,1112951
EC00632=798156,1112951
EC00633=798154,1112949
EC00634=798156,1112951
EC00635=798156,1112951
EC00636=798154,1112949
EC00637=798154,1112949
EC00638=798154,1112949
EC00639=798154,1112949
EC00640=798154,1112949
EC00641=798154,1112949
EC00642=798156,1112951
EC00643=798156,1112951
EC00644=798156,1112951
EC00645=798156,1112951
EC00646=798156,1112951
EC00647=798156,1112951
EC00648=798156,1112951
EC00649=798156,1112951
EC00650=798156,1112951
EC00651=798156,1112951
EC00652=798156,1112951
EC00653=798156,1112951
EC00654=798156,1112951
EC00655=798156,1112951
EC00656=798156,1112951
EC00657=798156,1112951
EC00658=798156,1112951
EC00659=798156,1112951
EC00660=798156,1112951
EC00661=798156,1112951
EC00662=798156,1112951
EC00663=798156,1112951
EC00664=798156,1112951
EC00665=798156,1112951
EC00666=798156,1112951
EC00667=798156,1112951
EC00668=798156,1112951
EC00669=798156,1112951
EC00670=798156,1112951
EC00671=798156,1112951
EC00672=798156,1112951
EC00673=798155,1112950
EC00674=798155,1112950
///POSTYPE BASE
///RECTAN
///RCONF 0,0,0,0,0,0,0,0,0,0,0,0,0,0,0,0,0,0,0,0,0,0,0,0
P00006=0.222,-3.123,-1.508,0.0000,0.0000,0.0000
P00021=-0.225,-6.128,-0.405,0.0000,0.0000,0.0000
P00022=0.222,-3.123,-1.508,0.0000,0.0000,0.0000
P00023=0.143,-0.036,0.682,0.0000,0.0000,0.0000
P00030=5.926,-4.294,-1.390,0.0000,0.0000,0.0000
P00031=1.853,-0.001,-1.549,0.0000,0.0000,0.0000
P00032=1.957,0.503,-7.217,0.0000,0.0000,0.0000
///RCONF 0,0,0,0,1,0,0,0,0,0,0,0,0,0,0,0,0,0,0,0,0,0,0,0
P00033=-0.123,0.612,-5.012,0.0000,0.0000,0.0000
///RCONF 0,0,0,0,0,0,0,0,0,0,0,0,0,0,0,0,0,0,0,0,0,0,0,0
P00034=-0.304,0.773,-2.693,0.0000,0.0000,0.0000
P00035=2.817,0.591,-1.622,0.0000,0.0000,0.0000
P00036=-1.108,-0.829,1.850,0.0000,0.0000,0.0000
P00037=0.023,0.937,-2.677,0.0000,0.0000,0.0000
P00038=0.158,-1.133,-1.952,0.0000,0.0000,0.0000
P00039=0.012,-3.081,-0.106,0.0000,0.0000,0.0000
P00040=-0.030,9.648,2.467,0.0000,0.0000,0.0000
P00041=0.192,3.924,0.305,0.0000,0.0000,0.0000
P00042=-0.217,1.941,0.413,0.0000,0.0000,0.0000
P00043=-0.044,-1.937,1.197,0.0000,0.0000,0.0000
P00044=0.687,-2.322,1.156,0.0000,0.0000,0.0000
//INST
///DATE 2025/03/04 13:38
///ATTR SC,RW
///GROUP1 RB1,BS1
///GROUP2 ST1
NOP
'OK_r2_O38-47,64(1)(90,180)
'Down
MOVJ C00000 BC00000 VJ=100.00  +MOVJ EC00000 VJ=100.00
MOVJ C00001 BC00001 VJ=100.00  +MOVJ EC00001 VJ=100.00
MOVJ C00002 BC00002 VJ=100.00  +MOVJ EC00002 VJ=100.00
'Path S1883
SFTOF3D
MOVJ C00003 BC00003 VJ=100.00  +MOVJ EC00003 VJ=100.00
MOVL C00004 BC00004 V=500.0  +MOVJ EC00004 VJ=100.00
SMOVL C00005 BC00005 V=100.0  +MOVJ EC00005
SREFP 3 C00006 BC00006  +REFP EC00006
CALL JOB:SEARCH-R1-S13D
SET P021 P006
SFTON3D P021
SMOVL C00007 BC00007 V=100.0  +MOVJ EC00007
SMOVL C00008 BC00008 V=100.0  +MOVJ EC00008
SMOVL C00009 BC00009 V=100.0  +MOVJ EC00009
SREFP 3 C00010 BC00010  +REFP EC00010
CALL JOB:SEARCH-R1-S13D
SET P021 P006
SFTON3D P021
SMOVL C00011 BC00011 V=100.0  +MOVJ EC00011
MOVL C00012 BC00012 V=400.0  +MOVJ EC00012 VJ=100.00
MOVJ C00013 BC00013 VJ=100.00  +MOVJ EC00013 VJ=100.00
MOVJ C00014 BC00014 VJ=100.00  +MOVJ EC00014 VJ=100.00
MOVJ C00015 BC00015 VJ=100.00  +MOVJ EC00015 VJ=100.00
MOVJ C00016 BC00016 VJ=100.00  +MOVJ EC00016 VJ=100.00
'Path S1884
SFTOF3D
MOVJ C00017 BC00017 VJ=40.00  +MOVJ EC00017 VJ=100.00
MOVL C00018 BC00018 V=400.0  +MOVJ EC00018 VJ=100.00
SMOVL C00019 BC00019 V=100.0  +MOVJ EC00019
SREFP 3 C00020 BC00020  +REFP EC00020
CALL JOB:SEARCH-R1-S13D
SET P022 P006
SFTON3D P022
SMOVL C00021 BC00021 V=100.0  +MOVJ EC00021
SMOVL C00022 BC00022 V=133.3  +MOVJ EC00022
SMOVL C00023 BC00023 V=100.0  +MOVJ EC00023
SREFP 3 C00024 BC00024  +REFP EC00024
CALL JOB:SEARCH-R1-S13D
SET P022 P006
SFTON3D P022
SMOVL C00025 BC00025 V=100.0  +MOVJ EC00025
MOVL C00026 BC00026 V=1000.0  +MOVJ EC00026 VJ=100.00
MOVJ C00027 BC00027 VJ=100.00  +MOVJ EC00027 VJ=100.00
MOVJ C00028 BC00028 VJ=100.00  +MOVJ EC00028 VJ=100.00
MOVJ C00029 BC00029 VJ=100.00  +MOVJ EC00029 VJ=100.00
MOVJ C00030 BC00030 VJ=100.00  +MOVJ EC00030 VJ=100.00
MOVJ C00031 BC00031 VJ=100.00  +MOVJ EC00031 VJ=100.00
'Path S1885
SFTOF3D
MOVJ C00032 BC00032 VJ=100.00  +MOVJ EC00032 VJ=100.00
MOVL C00033 BC00033 V=166.7  +MOVJ EC00033 VJ=100.00
SMOVL C00034 BC00034 V=100.0  +MOVJ EC00034
SREFP 3 C00035 BC00035  +REFP EC00035
CALL JOB:SEARCH-R1-S13D
SET P023 P006
SFTON3D P023
SMOVL C00036 BC00036 V=100.0  +MOVJ EC00036
SMOVL C00037 BC00037 V=166.7  +MOVJ EC00037
SMOVL C00038 BC00038 V=100.0  +MOVJ EC00038
SREFP 3 C00039 BC00039  +REFP EC00039
CALL JOB:SEARCH-R1-S13D
SET P023 P006
SFTON3D P023
SMOVL C00040 BC00040 V=100.0  +MOVJ EC00040
SFTOF3D
MOVL C00041 BC00041 V=400.0  +MOVJ EC00041 VJ=100.00
MOVL C00042 BC00042 V=1000.0  +MOVJ EC00042 VJ=100.00
MOVL C00043 BC00043 V=1000.0  +MOVJ EC00043 VJ=100.00
MOVJ C00044 BC00044 VJ=100.00  +MOVJ EC00044 VJ=100.00
MOVJ C00045 BC00045 VJ=100.00  +MOVJ EC00045 VJ=100.00
MOVJ C00046 BC00046 VJ=100.00  +MOVJ EC00046 VJ=100.00
'NOWY PROGRAM KRIS
MOVJ C00047 BC00047 VJ=100.00  +MOVJ EC00047 VJ=100.00
MOVJ C00048 BC00048 VJ=100.00  +MOVJ EC00048 VJ=100.00
MOVJ C00049 BC00049 VJ=100.00  +MOVJ EC00049 VJ=100.00
COMM PAUSE
COMM SMOVL C00050 BC00050 V=100.0  +MOVJ EC00050
COMM SREFP 3 C00051 BC00051  +REFP EC00051
COMM CALL JOB:SEARCH-R1-S13D
COMM SET P030 P006
COMM SFTON3D P030
COMM SMOVL C00052 BC00052 V=100.0  +MOVJ EC00052
COMM SREFP 3 C00053 BC00053  +REFP EC00053
COMM CALL JOB:SEARCH-R1-S13D
COMM SET P030 P006
COMM SFTON3D P030
COMM SMOVL C00054 BC00054 V=100.0  +MOVJ EC00054
COMM SFTOF3D
COMM MOVJ C00055 BC00055 VJ=100.00  +MOVJ EC00055 VJ=100.00
COMM SMOVL C00056 BC00056 V=100.0  +MOVJ EC00056
COMM SREFP 3 C00057 BC00057  +REFP EC00057
COMM CALL JOB:SEARCH-R1-S13D
COMM SET P031 P006
COMM SFTON3D P031
COMM SMOVL C00058 BC00058 V=100.0  +MOVJ EC00058
COMM SREFP 3 C00059 BC00059  +REFP EC00059
COMM CALL JOB:SEARCH-R1-S13D
COMM SET P031 P006
COMM SFTON3D P031
COMM SMOVL C00060 BC00060 V=100.0  +MOVJ EC00060
COMM SFTOF3D
MOVJ C00061 BC00061 VJ=100.00  +MOVJ EC00061 VJ=100.00
MOVJ C00062 BC00062 VJ=100.00  +MOVJ EC00062 VJ=100.00
MOVJ C00063 BC00063 VJ=100.00  +MOVJ EC00063 VJ=100.00
SMOVL C00064 BC00064 V=100.0  +MOVJ EC00064
SREFP 3 C00065 BC00065  +REFP EC00065
CALL JOB:SEARCH-R1-S13D
SET P032 P006
SFTON3D P032
SMOVL C00066 BC00066 V=100.0  +MOVJ EC00066
SREFP 3 C00067 BC00067  +REFP EC00067
CALL JOB:SEARCH-R1-S13D
SET P032 P006
SFTON3D P032
SMOVL C00068 BC00068 V=100.0  +MOVJ EC00068
SFTOF3D
MOVJ C00069 BC00069 VJ=100.00  +MOVJ EC00069 VJ=100.00
SMOVL C00070 BC00070 V=100.0  +MOVJ EC00070
SREFP 3 C00071 BC00071  +REFP EC00071
CALL JOB:SEARCH-R1-S13D
SET P033 P006
SFTON3D P033
SMOVL C00072 BC00072 V=100.0  +MOVJ EC00072
SREFP 3 C00073 BC00073  +REFP EC00073
CALL JOB:SEARCH-R1-S13D
SET P033 P006
SFTON3D P033
SMOVL C00074 BC00074 V=100.0  +MOVJ EC00074
SFTOF3D
MOVJ C00075 BC00075 VJ=100.00  +MOVJ EC00075 VJ=100.00
MOVJ C00076 BC00076 VJ=100.00  +MOVJ EC00076 VJ=100.00
SMOVL C00077 BC00077 V=100.0  +MOVJ EC00077
SREFP 3 C00078 BC00078  +REFP EC00078
CALL JOB:SEARCH-R1-S13D
SET P034 P006
SFTON3D P034
SMOVL C00079 BC00079 V=100.0  +MOVJ EC00079
SREFP 3 C00080 BC00080  +REFP EC00080
CALL JOB:SEARCH-R1-S13D
SET P034 P006
SFTON3D P034
SMOVL C00081 BC00081 V=100.0  +MOVJ EC00081
SFTOF3D
MOVJ C00082 BC00082 VJ=100.00  +MOVJ EC00082 VJ=100.00
MOVJ C00083 BC00083 VJ=100.00  +MOVJ EC00083 VJ=100.00
MOVJ C00084 BC00084 VJ=100.00  +MOVJ EC00084 VJ=100.00
SMOVL C00085 BC00085 V=100.0  +MOVJ EC00085
SREFP 3 C00086 BC00086  +REFP EC00086
CALL JOB:SEARCH-R1-S13D
SET P035 P006
SFTON3D P035
SMOVL C00087 BC00087 V=100.0  +MOVJ EC00087
SREFP 3 C00088 BC00088  +REFP EC00088
CALL JOB:SEARCH-R1-S13D
SET P035 P006
SFTON3D P035
SMOVL C00089 BC00089 V=100.0  +MOVJ EC00089
SFTOF3D
MOVJ C00090 BC00090 VJ=100.00  +MOVJ EC00090 VJ=100.00
SMOVL C00091 BC00091 V=100.0  +MOVJ EC00091
SREFP 3 C00092 BC00092  +REFP EC00092
CALL JOB:SEARCH-R1-S13D
SET P036 P006
SFTON3D P036
SMOVL C00093 BC00093 V=100.0  +MOVJ EC00093
SREFP 3 C00094 BC00094  +REFP EC00094
CALL JOB:SEARCH-R1-S13D
SET P036 P006
SFTON3D P036
SMOVL C00095 BC00095 V=100.0  +MOVJ EC00095
SFTOF3D
MOVJ C00096 BC00096 VJ=100.00  +MOVJ EC00096 VJ=100.00
MOVJ C00097 BC00097 VJ=100.00  +MOVJ EC00097 VJ=100.00
MOVJ C00098 BC00098 VJ=100.00  +MOVJ EC00098 VJ=100.00
SMOVL C00099 BC00099 V=100.0  +MOVJ EC00099
SREFP 3 C00100 BC00100  +REFP EC00100
CALL JOB:SEARCH-R1-S13D
SET P044 P006
SFTON3D P044
SMOVL C00101 BC00101 V=100.0  +MOVJ EC00101
SREFP 3 C00102 BC00102  +REFP EC00102
CALL JOB:SEARCH-R1-S13D
SET P044 P006
SFTON3D P044
SMOVL C00103 BC00103 V=100.0  +MOVJ EC00103
SFTOF3D
MOVJ C00104 BC00104 VJ=100.00  +MOVJ EC00104 VJ=100.00
MOVJ C00105 BC00105 VJ=100.00  +MOVJ EC00105 VJ=100.00
COMM PAUSE
COMM MOVJ C00106 BC00106 VJ=100.00  +MOVJ EC00106 VJ=100.00
COMM MOVJ C00107 BC00107 VJ=100.00  +MOVJ EC00107 VJ=100.00
COMM SMOVL C00108 BC00108 V=100.0  +MOVJ EC00108
COMM SREFP 3 C00109 BC00109  +REFP EC00109
COMM CALL JOB:SEARCH-R1-S13D
COMM SET P037 P006
COMM SFTON3D P037
COMM SMOVL C00110 BC00110 V=100.0  +MOVJ EC00110
COMM SREFP 3 C00111 BC00111  +REFP EC00111
COMM CALL JOB:SEARCH-R1-S13D
COMM SET P037 P006
COMM SFTON3D P037
COMM SMOVL C00112 BC00112 V=100.0  +MOVJ EC00112
COMM SFTOF3D
COMM MOVJ C00113 BC00113 VJ=100.00  +MOVJ EC00113 VJ=100.00
COMM SMOVL C00114 BC00114 V=100.0  +MOVJ EC00114
COMM SREFP 3 C00115 BC00115  +REFP EC00115
COMM CALL JOB:SEARCH-R1-S13D
COMM SET P038 P006
COMM SFTON3D P038
COMM SMOVL C00116 BC00116 V=100.0  +MOVJ EC00116
COMM SREFP 3 C00117 BC00117  +REFP EC00117
COMM CALL JOB:SEARCH-R1-S13D
COMM SET P038 P006
COMM SFTON3D P038
COMM SMOVL C00118 BC00118 V=100.0  +MOVJ EC00118
COMM SFTOF3D
COMM MOVJ C00119 BC00119 VJ=100.00  +MOVJ EC00119 VJ=100.00
MOVJ C00120 BC00120 VJ=100.00  +MOVJ EC00120 VJ=100.00
MOVJ C00121 BC00121 VJ=100.00  +MOVJ EC00121 VJ=100.00
MOVJ C00122 BC00122 VJ=100.00  +MOVJ EC00122 VJ=100.00
SMOVL C00123 BC00123 V=100.0  +MOVJ EC00123
SREFP 3 C00124 BC00124  +REFP EC00124
CALL JOB:SEARCH-R1-S13D
SET P039 P006
SFTON3D P039
SMOVL C00125 BC00125 V=100.0  +MOVJ EC00125
SREFP 3 C00126 BC00126  +REFP EC00126
CALL JOB:SEARCH-R1-S13D
SET P039 P006
SFTON3D P039
SMOVL C00127 BC00127 V=100.0  +MOVJ EC00127
SFTOF3D
MOVJ C00128 BC00128 VJ=100.00  +MOVJ EC00128 VJ=100.00
SMOVL C00129 BC00129 V=100.0  +MOVJ EC00129
SREFP 3 C00130 BC00130  +REFP EC00130
CALL JOB:SEARCH-R1-S13D
SET P040 P006
SFTON3D P040
SMOVL C00131 BC00131 V=100.0  +MOVJ EC00131
SREFP 3 C00132 BC00132  +REFP EC00132
CALL JOB:SEARCH-R1-S13D
SET P040 P006
SFTON3D P040
SMOVL C00133 BC00133 V=100.0  +MOVJ EC00133
MOVJ C00134 BC00134 VJ=100.00  +MOVJ EC00134 VJ=100.00
SFTOF3D
MOVJ C00135 BC00135 VJ=100.00  +MOVJ EC00135 VJ=100.00
MOVJ C00136 BC00136 VJ=100.00  +MOVJ EC00136 VJ=100.00
SMOVL C00137 BC00137 V=100.0  +MOVJ EC00137
SREFP 3 C00138 BC00138  +REFP EC00138
CALL JOB:SEARCH-R1-S13D
SET P041 P006
SFTON3D P041
SMOVL C00139 BC00139 V=100.0  +MOVJ EC00139
SREFP 3 C00140 BC00140  +REFP EC00140
CALL JOB:SEARCH-R1-S13D
SET P041 P006
SFTON3D P041
SMOVL C00141 BC00141 V=100.0  +MOVJ EC00141
SFTOF3D
MOVJ C00142 BC00142 VJ=100.00  +MOVJ EC00142 VJ=100.00
SMOVL C00143 BC00143 V=100.0  +MOVJ EC00143
SREFP 3 C00144 BC00144  +REFP EC00144
CALL JOB:SEARCH-R1-S13D
SET P042 P006
SFTON3D P042
SMOVL C00145 BC00145 V=100.0  +MOVJ EC00145
SREFP 3 C00146 BC00146  +REFP EC00146
CALL JOB:SEARCH-R1-S13D
SET P042 P006
SFTON3D P042
SMOVL C00147 BC00147 V=250.0  +MOVJ EC00147
MOVJ C00148 BC00148 VJ=100.00  +MOVJ EC00148 VJ=100.00
SFTOF3D
MOVJ C00149 BC00149 VJ=100.00  +MOVJ EC00149 VJ=100.00
SMOVL C00150 BC00150 V=100.0  +MOVJ EC00150
SREFP 3 C00151 BC00151  +REFP EC00151
CALL JOB:SEARCH-R1-S13D
SET P043 P006
SFTON3D P043
SMOVL C00152 BC00152 V=100.0  +MOVJ EC00152
SREFP 3 C00153 BC00153  +REFP EC00153
CALL JOB:SEARCH-R1-S13D
SET P043 P006
SFTON3D P043
SMOVL C00154 BC00154 V=166.7  +MOVJ EC00154
'KONIEC POMIARU
SMOVL C00155 BC00155 V=166.7  +MOVJ EC00155
MACRO1 MJ#(0) ARGF9
SFTON3D P043
SMOVL C00156 BC00156 V=250.0  +MOVJ EC00156
ARCON
SWVON WEV#(30)
SMOVL C00157 BC00157 V=10.0  +MOVJ EC00157
SMOVL C00158 BC00158 V=10.0  +MOVJ EC00158
SMOVL C00159 BC00159 V=10.0  +MOVJ EC00159
ARCOF
SWVOF
SFTOF3D
MOVJ C00160 BC00160 VJ=15.00  +MOVJ EC00160 VJ=100.00
MOVJ C00161 BC00161 VJ=100.00  +MOVJ EC00161 VJ=100.00
MOVJ C00162 BC00162 VJ=100.00  +MOVJ EC00162 VJ=100.00
MOVJ C00163 BC00163 VJ=100.00  +MOVJ EC00163 VJ=100.00
SFTON3D P044
SMOVL C00164 BC00164 V=166.7 PL=0  +MOVJ EC00164
ARCON
SWVON WEV#(30)
SMOVL C00165 BC00165 V=8.3  +MOVJ EC00165
SMOVL C00166 BC00166 V=8.3  +MOVJ EC00166
SMOVL C00167 BC00167 V=8.3  +MOVJ EC00167
ARCOF
SWVOF
SFTOF3D
MOVJ C00168 BC00168 VJ=15.00  +MOVJ EC00168 VJ=15.00
COMM PAUSE
COMM MOVJ C00169 BC00169 VJ=100.00  +MOVJ EC00169 VJ=100.00
COMM MACRO1 MJ#(0) ARGF9
COMM SFTON3D P031
COMM SMOVL C00170 BC00170 V=133.3  +MOVJ EC00170
COMM ARCON
COMM SWVON WEV#(10)
COMM SMOVL C00171 BC00171 V=10.0  +MOVJ EC00171
COMM SFTON3D P030
COMM SMOVL C00172 BC00172 V=10.0  +MOVJ EC00172
COMM SMOVL C00173 BC00173 V=10.0  +MOVJ EC00173
COMM ARCOF
COMM SWVOF
COMM SFTOF
COMM MOVJ C00174 BC00174 VJ=100.00  +MOVJ EC00174 VJ=100.00
COMM MOVJ C00175 BC00175 VJ=100.00  +MOVJ EC00175 VJ=100.00
COMM MOVJ C00176 BC00176 VJ=100.00  +MOVJ EC00176 VJ=100.00
COMM SFTON3D P038
COMM SMOVL C00177 BC00177 V=166.7  +MOVJ EC00177
COMM ARCON
COMM SFTON3D P037
COMM MOVL C00178 BC00178 V=9.2  +MOVJ EC00178 VJ=100.00
COMM ARCOF
COMM TIMER T=1.00
COMM SFTOF3D
COMM MOVJ C00179 BC00179 VJ=100.00  +MOVJ EC00179 VJ=100.00
COMM MOVJ C00180 BC00180 VJ=100.00  +MOVJ EC00180 VJ=100.00
COMM MOVJ C00181 BC00181 VJ=100.00  +MOVJ EC00181 VJ=100.00
MOVJ C00182 BC00182 VJ=100.00  +MOVJ EC00182 VJ=100.00
MACRO1 MJ#(0) ARGF14
MOVJ C00183 BC00183 VJ=100.00  +MOVJ EC00183 VJ=100.00
SFTON3D P041
SMOVL C00184 BC00184 V=166.7  +MOVJ EC00184
ARCON
SMOVL C00185 BC00185 V=9.2  +MOVJ EC00185
SFTON3D P042
SMOVL C00186 BC00186 V=9.2  +MOVJ EC00186
ARCOF
SFTOF3D
MOVJ C00187 BC00187 VJ=100.00  +MOVJ EC00187 VJ=100.00
MOVJ C00188 BC00188 VJ=100.00  +MOVJ EC00188 VJ=100.00
SFTON3D P040
SMOVL C00189 BC00189 V=166.7  +MOVJ EC00189
ARCON
SMOVL C00190 BC00190 V=9.2  +MOVJ EC00190
SFTON3D P039
SMOVL C00191 BC00191 V=9.2  +MOVJ EC00191
SMOVL C00192 BC00192 V=9.2  +MOVJ EC00192
ARCOF
MOVJ C00193 BC00193 VJ=100.00  +MOVJ EC00193 VJ=100.00
MOVJ C00194 BC00194 VJ=100.00  +MOVJ EC00194 VJ=100.00
MOVJ C00195 BC00195 VJ=100.00  +MOVJ EC00195 VJ=100.00
MOVJ C00196 BC00196 VJ=100.00  +MOVJ EC00196 VJ=100.00
MACRO1 MJ#(0) ARGF9
SFTON3D P036
SMOVL C00197 BC00197 V=166.7  +MOVJ EC00197
ARCON
SMOVL C00198 BC00198 V=9.2  +MOVJ EC00198
SFTON3D P035
SMOVL C00199 BC00199 V=9.2  +MOVJ EC00199
SMOVL C00200 BC00200 V=9.2  +MOVJ EC00200
ARCOF
SFTOF3D
MOVJ C00201 BC00201 VJ=15.00  +MOVJ EC00201 VJ=100.00
MOVJ C00202 BC00202 VJ=100.00  +MOVJ EC00202 VJ=15.00
MACRO1 MJ#(0) ARGF9
SFTON3D P034
SMOVL C00203 BC00203 V=166.7  +MOVJ EC00203
ARCON
SMOVC C00204 BC00204 V=8.3  +MOVJ EC00204
SMOVC C00205 BC00205 V=8.3  +MOVJ EC00205
SMOVC C00206 BC00206 V=8.3  +MOVJ EC00206
SMOVL C00207 BC00207 V=10.0  +MOVJ EC00207
SMOVC C00208 BC00208 V=8.3  +MOVJ EC00208
SMOVC C00209 BC00209 V=8.3  +MOVJ EC00209
SMOVC C00210 BC00210 V=8.3  +MOVJ EC00210
ARCOF
SFTOF3D
MOVJ C00211 BC00211 VJ=100.00  +MOVJ EC00211 VJ=100.00
MOVJ C00212 BC00212 VJ=100.00  +MOVJ EC00212 VJ=100.00
SFTON3D P032
SMOVL C00213 BC00213 V=250.0  +MOVJ EC00213
ARCON
SMOVL C00214 BC00214 V=8.3  +MOVJ EC00214
SFTON3D P033
SMOVL C00215 BC00215 V=8.3  +MOVJ EC00215
SMOVL C00216 BC00216 V=8.3  +MOVJ EC00216
ARCOF
SFTOF3D
MOVJ C00217 BC00217 VJ=30.00  +MOVJ EC00217 VJ=100.00
MOVJ C00218 BC00218 VJ=30.00  +MOVJ EC00218 VJ=15.00
JUMP *LABEL
'Up
'Path S1856
SFTOF3D
MOVJ C00219 BC00219 VJ=100.00  +MOVJ EC00219 VJ=100.00
COMM MOVL C00220 BC00220 V=400.0  +MOVJ EC00220 VJ=100.00
COMM SMOVL C00221 BC00221 V=60.0  +MOVJ EC00221
COMM SREFP 3 C00222 BC00222  +REFP EC00222
COMM CALL JOB:SEARCH-R1-S13D
COMM SET P042 P006
COMM SFTON3D P042
COMM SMOVL C00223 BC00223 V=60.0  +MOVJ EC00223
COMM SMOVL C00224 BC00224 V=60.0  +MOVJ EC00224
COMM SREFP 3 C00225 BC00225  +REFP EC00225
COMM CALL JOB:SEARCH-R1-S13D
COMM SET P042 P006
COMM SFTON3D P042
COMM SMOVL C00226 BC00226 V=60.0  +MOVJ EC00226
COMM MOVL C00227 BC00227 V=400.0  +MOVJ EC00227 VJ=100.00
COMM MOVL C00228 BC00228 V=1000.0  +MOVJ EC00228 VJ=100.00
COMM 'Path S1857
COMM SFTOF3D
COMM MOVJ C00229 BC00229 VJ=100.00  +MOVJ EC00229 VJ=100.00
COMM MOVL C00230 BC00230 V=400.0  +MOVJ EC00230 VJ=100.00
COMM SMOVL C00231 BC00231 V=60.0  +MOVJ EC00231
COMM SREFP 3 C00232 BC00232  +REFP EC00232
COMM CALL JOB:SEARCH-R1-S13D
COMM SET P041 P006
COMM SFTON3D P041
COMM SMOVL C00233 BC00233 V=60.0  +MOVJ EC00233
COMM SMOVL C00234 BC00234 V=60.0  +MOVJ EC00234
COMM SREFP 3 C00235 BC00235  +REFP EC00235
COMM CALL JOB:SEARCH-R1-S13D
COMM SET P041 P006
COMM SFTON3D P041
COMM SMOVL C00236 BC00236 V=60.0  +MOVJ EC00236
COMM MOVL C00237 BC00237 V=400.0  +MOVJ EC00237 VJ=100.00
COMM MOVL C00238 BC00238 V=1000.0  +MOVJ EC00238 VJ=100.00
COMM 'Path S1858
COMM SFTOF3D
COMM MOVJ C00239 BC00239 VJ=100.00  +MOVJ EC00239 VJ=100.00
COMM MOVL C00240 BC00240 V=400.0  +MOVJ EC00240 VJ=100.00
COMM SMOVL C00241 BC00241 V=60.0  +MOVJ EC00241
COMM SREFP 3 C00242 BC00242  +REFP EC00242
COMM CALL JOB:SEARCH-R1-S13D
COMM SET P040 P006
COMM SFTON3D P040
COMM SMOVL C00243 BC00243 V=60.0  +MOVJ EC00243
COMM SMOVL C00244 BC00244 V=60.0  +MOVJ EC00244
COMM SREFP 3 C00245 BC00245  +REFP EC00245
COMM CALL JOB:SEARCH-R1-S13D
COMM SET P040 P006
COMM SFTON3D P040
COMM SMOVL C00246 BC00246 V=60.0  +MOVJ EC00246
COMM MOVL C00247 BC00247 V=400.0  +MOVJ EC00247 VJ=100.00
COMM MOVL C00248 BC00248 V=1000.0  +MOVJ EC00248 VJ=100.00
MOVL C00249 BC00249 V=1000.0  +MOVJ EC00249 VJ=100.00
'Path S1859
SFTOF3D
MOVJ C00250 BC00250 VJ=100.00  +MOVJ EC00250 VJ=100.00
MOVJ C00251 BC00251 VJ=100.00  +MOVJ EC00251 VJ=100.00
MOVL C00252 BC00252 V=400.0  +MOVJ EC00252 VJ=100.00
SMOVL C00253 BC00253 V=60.0  +MOVJ EC00253
SREFP 3 C00254 BC00254  +REFP EC00254
CALL JOB:SEARCH-R1-S13D
SET P043 P006
SFTON3D P043
SMOVL C00255 BC00255 V=60.0  +MOVJ EC00255
SMOVL C00256 BC00256 V=60.0  +MOVJ EC00256
SREFP 3 C00257 BC00257  +REFP EC00257
CALL JOB:SEARCH-R1-S13D
SET P043 P006
SFTON3D P043
SMOVL C00258 BC00258 V=60.0  +MOVJ EC00258
MOVL C00259 BC00259 V=400.0  +MOVJ EC00259 VJ=100.00
MOVL C00260 BC00260 V=1000.0  +MOVJ EC00260 VJ=100.00
'Path S1860
SFTOF3D
MOVJ C00261 BC00261 VJ=100.00  +MOVJ EC00261 VJ=100.00
MOVL C00262 BC00262 V=400.0  +MOVJ EC00262 VJ=100.00
SMOVL C00263 BC00263 V=60.0  +MOVJ EC00263
SREFP 3 C00264 BC00264  +REFP EC00264
CALL JOB:SEARCH-R1-S13D
SET P039 P006
SFTON3D P039
SMOVL C00265 BC00265 V=60.0  +MOVJ EC00265
SMOVL C00266 BC00266 V=60.0  +MOVJ EC00266
SREFP 3 C00267 BC00267  +REFP EC00267
CALL JOB:SEARCH-R1-S13D
SET P039 P006
SFTON3D P039
SMOVL C00268 BC00268 V=60.0  +MOVJ EC00268
MOVL C00269 BC00269 V=400.0  +MOVJ EC00269 VJ=100.00
MOVL C00270 BC00270 V=1000.0  +MOVJ EC00270 VJ=100.00
MOVJ C00271 BC00271 VJ=100.00  +MOVJ EC00271 VJ=100.00
'Path S1861
SFTOF3D
MOVJ C00272 BC00272 VJ=100.00  +MOVJ EC00272 VJ=100.00
MOVL C00273 BC00273 V=400.0  +MOVJ EC00273 VJ=100.00
SMOVL C00274 BC00274 V=60.0  +MOVJ EC00274
SREFP 3 C00275 BC00275  +REFP EC00275
CALL JOB:SEARCH-R1-S13D
SET P034 P006
SFTON3D P034
SMOVL C00276 BC00276 V=60.0  +MOVJ EC00276
SMOVL C00277 BC00277 V=60.0  +MOVJ EC00277
SREFP 3 C00278 BC00278  +REFP EC00278
CALL JOB:SEARCH-R1-S13D
SET P034 P006
SFTON3D P034
SMOVL C00279 BC00279 V=60.0  +MOVJ EC00279
MOVL C00280 BC00280 V=400.0  +MOVJ EC00280 VJ=100.00
MOVL C00281 BC00281 V=1000.0  +MOVJ EC00281 VJ=100.00
MOVJ C00282 BC00282 VJ=100.00  +MOVJ EC00282 VJ=100.00
'Path S1862
SFTOF3D
MOVJ C00283 BC00283 VJ=100.00  +MOVJ EC00283 VJ=100.00
MOVL C00284 BC00284 V=400.0  +MOVJ EC00284 VJ=100.00
SMOVL C00285 BC00285 V=60.0  +MOVJ EC00285
SREFP 3 C00286 BC00286  +REFP EC00286
CALL JOB:SEARCH-R1-S13D
SET P038 P006
SFTON3D P038
SMOVL C00287 BC00287 V=60.0  +MOVJ EC00287
SMOVL C00288 BC00288 V=60.0  +MOVJ EC00288
SREFP 3 C00289 BC00289  +REFP EC00289
CALL JOB:SEARCH-R1-S13D
SET P038 P006
SFTON3D P038
SMOVL C00290 BC00290 V=60.0  +MOVJ EC00290
SMOVL C00291 BC00291 V=60.0  +MOVJ EC00291
SREFP 3 C00292 BC00292  +REFP EC00292
CALL JOB:SEARCH-R1-S13D
SET P038 P006
SFTON3D P038
SMOVL C00293 BC00293 V=60.0  +MOVJ EC00293
MOVL C00294 BC00294 V=400.0  +MOVJ EC00294 VJ=100.00
MOVL C00295 BC00295 V=1000.0  +MOVJ EC00295 VJ=100.00
'Path S1863
SFTOF3D
MOVJ C00296 BC00296 VJ=100.00  +MOVJ EC00296 VJ=100.00
MOVL C00297 BC00297 V=400.0  +MOVJ EC00297 VJ=100.00
SMOVL C00298 BC00298 V=60.0  +MOVJ EC00298
SREFP 3 C00299 BC00299  +REFP EC00299
CALL JOB:SEARCH-R1-S13D
SET P033 P006
SFTON3D P033
SMOVL C00300 BC00300 V=60.0  +MOVJ EC00300
SMOVL C00301 BC00301 V=60.0  +MOVJ EC00301
SREFP 3 C00302 BC00302  +REFP EC00302
CALL JOB:SEARCH-R1-S13D
SET P033 P006
SFTON3D P033
SMOVL C00303 BC00303 V=60.0  +MOVJ EC00303
MOVL C00304 BC00304 V=400.0  +MOVJ EC00304 VJ=100.00
MOVL C00305 BC00305 V=1000.0  +MOVJ EC00305 VJ=100.00
MOVL C00306 BC00306 V=1000.0  +MOVJ EC00306 VJ=100.00
'Path S1864
SFTOF3D
MOVJ C00307 BC00307 VJ=100.00  +MOVJ EC00307 VJ=100.00
MOVJ C00308 BC00308 VJ=100.00  +MOVJ EC00308 VJ=100.00
MOVL C00309 BC00309 V=400.0  +MOVJ EC00309 VJ=100.00
SMOVL C00310 BC00310 V=60.0  +MOVJ EC00310
SREFP 3 C00311 BC00311  +REFP EC00311
CALL JOB:SEARCH-R1-S13D
SET P035 P006
SFTON3D P035
SMOVL C00312 BC00312 V=60.0  +MOVJ EC00312
SMOVL C00313 BC00313 V=60.0  +MOVJ EC00313
SREFP 3 C00314 BC00314  +REFP EC00314
CALL JOB:SEARCH-R1-S13D
SET P035 P006
SFTON3D P035
SMOVL C00315 BC00315 V=60.0  +MOVJ EC00315
MOVL C00316 BC00316 V=400.0  +MOVJ EC00316 VJ=100.00
MOVL C00317 BC00317 V=1000.0  +MOVJ EC00317 VJ=100.00
MOVL C00318 BC00318 V=1000.0  +MOVJ EC00318 VJ=100.00
'Path S1865
SFTOF3D
MOVJ C00319 BC00319 VJ=100.00  +MOVJ EC00319 VJ=100.00
MOVL C00320 BC00320 V=400.0  +MOVJ EC00320 VJ=100.00
SMOVL C00321 BC00321 V=60.0  +MOVJ EC00321
SREFP 3 C00322 BC00322  +REFP EC00322
CALL JOB:SEARCH-R1-S13D
SET P037 P006
SFTON3D P037
SMOVL C00323 BC00323 V=60.0  +MOVJ EC00323
SMOVL C00324 BC00324 V=60.0  +MOVJ EC00324
SREFP 3 C00325 BC00325  +REFP EC00325
CALL JOB:SEARCH-R1-S13D
SET P037 P006
SFTON3D P037
SMOVL C00326 BC00326 V=60.0  +MOVJ EC00326
MOVL C00327 BC00327 V=400.0  +MOVJ EC00327 VJ=100.00
MOVL C00328 BC00328 V=1000.0  +MOVJ EC00328 VJ=100.00
'Path S1866
SFTOF3D
MOVJ C00329 BC00329 VJ=100.00  +MOVJ EC00329 VJ=100.00
MOVJ C00330 BC00330 VJ=100.00  +MOVJ EC00330 VJ=100.00
MOVL C00331 BC00331 V=400.0  +MOVJ EC00331 VJ=100.00
SMOVL C00332 BC00332 V=60.0  +MOVJ EC00332
SREFP 3 C00333 BC00333  +REFP EC00333
CALL JOB:SEARCH-R1-S13D
SET P031 P006
SFTON3D P031
SMOVL C00334 BC00334 V=60.0  +MOVJ EC00334
SMOVL C00335 BC00335 V=60.0  +MOVJ EC00335
SREFP 3 C00336 BC00336  +REFP EC00336
CALL JOB:SEARCH-R1-S13D
SET P031 P006
SFTON3D P031
SMOVL C00337 BC00337 V=60.0  +MOVJ EC00337
MOVL C00338 BC00338 V=400.0  +MOVJ EC00338 VJ=100.00
MOVL C00339 BC00339 V=1000.0  +MOVJ EC00339 VJ=100.00
'Path S1867
MOVJ C00340 BC00340 VJ=20.00  +MOVJ EC00340 VJ=20.00
MOVJ C00341 BC00341 VJ=20.00  +MOVJ EC00341 VJ=20.00
SFTOF3D
MOVJ C00342 BC00342 VJ=100.00  +MOVJ EC00342 VJ=100.00
MOVL C00343 BC00343 V=400.0  +MOVJ EC00343 VJ=100.00
SMOVL C00344 BC00344 V=60.0  +MOVJ EC00344
SREFP 3 C00345 BC00345  +REFP EC00345
CALL JOB:SEARCH-R1-S13D
SET P036 P006
SFTON3D P036
SMOVL C00346 BC00346 V=60.0  +MOVJ EC00346
SMOVL C00347 BC00347 V=60.0  +MOVJ EC00347
SREFP 3 C00348 BC00348  +REFP EC00348
CALL JOB:SEARCH-R1-S13D
SET P036 P006
SFTON3D P036
SMOVL C00349 BC00349 V=60.0  +MOVJ EC00349
MOVL C00350 BC00350 V=400.0  +MOVJ EC00350 VJ=100.00
MOVL C00351 BC00351 V=1000.0  +MOVJ EC00351 VJ=100.00
MOVL C00352 BC00352 V=1000.0  +MOVJ EC00352 VJ=100.00
'Path S1868
SFTOF3D
MOVJ C00353 BC00353 VJ=100.00  +MOVJ EC00353 VJ=100.00
MOVL C00354 BC00354 V=400.0  +MOVJ EC00354 VJ=100.00
SMOVL C00355 BC00355 V=60.0  +MOVJ EC00355
SREFP 3 C00356 BC00356  +REFP EC00356
CALL JOB:SEARCH-R1-S13D
SET P032 P006
SFTON3D P032
SMOVL C00357 BC00357 V=60.0  +MOVJ EC00357
SMOVL C00358 BC00358 V=60.0  +MOVJ EC00358
SREFP 3 C00359 BC00359  +REFP EC00359
CALL JOB:SEARCH-R1-S13D
SET P032 P006
SFTON3D P032
SMOVL C00360 BC00360 V=60.0  +MOVJ EC00360
MOVL C00361 BC00361 V=400.0  +MOVJ EC00361 VJ=100.00
MOVL C00362 BC00362 V=1000.0  +MOVJ EC00362 VJ=100.00
'Path W1869
SFTOF3D
SFTON3D P032
MOVJ C00363 BC00363 VJ=100.00  +MOVJ EC00363 VJ=100.00
SMOVL C00364 BC00364 V=400.0  +MOVJ EC00364
SMOVL C00365 BC00365 V=100.0 PL=0  +MOVJ EC00365
SREFP 1 C00366 BC00366  +REFP EC00366
SREFP 2 C00367 BC00367  +REFP EC00367
MACRO1 MJ#(0) ARGF0
ARCON
SMOVL C00368 BC00368 V=10.0  +MOVJ EC00368
SMOVL C00369 BC00369 V=10.0  +MOVJ EC00369
SMOVL C00370 BC00370 V=10.0  +MOVJ EC00370
ARCOF
SMOVL C00371 BC00371 V=400.0  +MOVJ EC00371
SMOVL C00372 BC00372 V=1000.0  +MOVJ EC00372
SMOVL C00373 BC00373 V=1000.0  +MOVJ EC00373
SFTOF3D
MOVJ C00374 BC00374 VJ=100.00  +MOVJ EC00374 VJ=100.00
'Path W1870
SFTOF3D
SFTON3D P033
MOVJ C00375 BC00375 VJ=100.00  +MOVJ EC00375 VJ=100.00
MOVJ C00376 BC00376 VJ=100.00  +MOVJ EC00376 VJ=100.00
SMOVL C00377 BC00377 V=400.0  +MOVJ EC00377
SMOVL C00378 BC00378 V=100.0 PL=0  +MOVJ EC00378
SREFP 1 C00379 BC00379  +REFP EC00379
SREFP 2 C00380 BC00380  +REFP EC00380
MACRO1 MJ#(0) ARGF0
ARCON
SMOVL C00381 BC00381 V=10.0  +MOVJ EC00381
SMOVL C00382 BC00382 V=10.0  +MOVJ EC00382
SMOVL C00383 BC00383 V=10.0  +MOVJ EC00383
ARCOF
SMOVL C00384 BC00384 V=400.0  +MOVJ EC00384
SMOVL C00385 BC00385 V=1000.0  +MOVJ EC00385
SFTOF3D
'Path W1871
SFTOF3D
SFTON3D P034
MOVJ C00386 BC00386 VJ=100.00  +MOVJ EC00386 VJ=100.00
SMOVL C00387 BC00387 V=400.0  +MOVJ EC00387
SMOVL C00388 BC00388 V=100.0 PL=0  +MOVJ EC00388
SREFP 1 C00389 BC00389  +REFP EC00389
SREFP 2 C00390 BC00390  +REFP EC00390
MACRO1 MJ#(0) ARGF0
ARCON
SMOVL C00391 BC00391 V=10.0  +MOVJ EC00391
SMOVL C00392 BC00392 V=10.0  +MOVJ EC00392
ARCOF
SMOVL C00393 BC00393 V=400.0  +MOVJ EC00393
SMOVL C00394 BC00394 V=1000.0  +MOVJ EC00394
SMOVL C00395 BC00395 V=1000.0  +MOVJ EC00395
SFTOF3D
MOVJ C00396 BC00396 VJ=20.00  +MOVJ EC00396 VJ=20.00
MOVJ C00397 BC00397 VJ=20.00  +MOVJ EC00397 VJ=20.00
'Path W1872
SFTOF3D
SFTON3D P031
MOVJ C00398 BC00398 VJ=100.00  +MOVJ EC00398 VJ=100.00
SMOVL C00399 BC00399 V=400.0  +MOVJ EC00399
SMOVL C00400 BC00400 V=100.0 PL=0  +MOVJ EC00400
SREFP 1 C00401 BC00401  +REFP EC00401
SREFP 2 C00402 BC00402  +REFP EC00402
MACRO1 MJ#(0) ARGF0
ARCON
SMOVL C00403 BC00403 V=10.0  +MOVJ EC00403
SMOVL C00404 BC00404 V=10.0  +MOVJ EC00404
ARCOF
SMOVL C00405 BC00405 V=400.0  +MOVJ EC00405
SMOVL C00406 BC00406 V=1000.0  +MOVJ EC00406
SMOVL C00407 BC00407 V=1000.0  +MOVJ EC00407
SFTOF3D
'Path W1873
MOVJ C00408 BC00408 VJ=20.00  +MOVJ EC00408 VJ=20.00
SFTOF3D
SFTON3D P035
MOVJ C00409 BC00409 VJ=100.00  +MOVJ EC00409 VJ=100.00
SMOVL C00410 BC00410 V=400.0  +MOVJ EC00410
SMOVL C00411 BC00411 V=100.0 PL=0  +MOVJ EC00411
SREFP 1 C00412 BC00412  +REFP EC00412
SREFP 2 C00413 BC00413  +REFP EC00413
MACRO1 MJ#(0) ARGF0
ARCON
SMOVL C00414 BC00414 V=10.0  +MOVJ EC00414
SMOVL C00415 BC00415 V=10.0  +MOVJ EC00415
ARCOF
SMOVL C00416 BC00416 V=400.0  +MOVJ EC00416
SMOVL C00417 BC00417 V=1000.0  +MOVJ EC00417
SMOVL C00418 BC00418 V=1000.0  +MOVJ EC00418
SFTOF3D
MOVJ C00419 BC00419 VJ=100.00  +MOVJ EC00419 VJ=100.00
'Path W1874
SFTOF3D
SFTON3D P036
MOVJ C00420 BC00420 VJ=100.00  +MOVJ EC00420 VJ=100.00
SMOVL C00421 BC00421 V=400.0  +MOVJ EC00421
SMOVL C00422 BC00422 V=100.0 PL=0  +MOVJ EC00422
SREFP 1 C00423 BC00423  +REFP EC00423
SREFP 2 C00424 BC00424  +REFP EC00424
MACRO1 MJ#(0) ARGF0
ARCON
SMOVL C00425 BC00425 V=10.0  +MOVJ EC00425
SMOVL C00426 BC00426 V=10.0  +MOVJ EC00426
SMOVL C00427 BC00427 V=10.0  +MOVJ EC00427
ARCOF
SMOVL C00428 BC00428 V=400.0  +MOVJ EC00428
SMOVL C00429 BC00429 V=1000.0  +MOVJ EC00429
SMOVL C00430 BC00430 V=1000.0  +MOVJ EC00430
SFTOF3D
MOVJ C00431 BC00431 VJ=100.00  +MOVJ EC00431 VJ=100.00
'Path W1875
SFTOF3D
SFTON3D P037
MOVJ C00432 BC00432 VJ=100.00  +MOVJ EC00432 VJ=100.00
MOVJ C00433 BC00433 VJ=100.00  +MOVJ EC00433 VJ=100.00
SMOVL C00434 BC00434 V=400.0  +MOVJ EC00434
SMOVL C00435 BC00435 V=100.0 PL=0  +MOVJ EC00435
SREFP 1 C00436 BC00436  +REFP EC00436
SREFP 2 C00437 BC00437  +REFP EC00437
MACRO1 MJ#(0) ARGF0
ARCON
SMOVL C00438 BC00438 V=10.0  +MOVJ EC00438
SMOVL C00439 BC00439 V=10.0  +MOVJ EC00439
SMOVL C00440 BC00440 V=10.0  +MOVJ EC00440
ARCOF
SMOVL C00441 BC00441 V=400.0  +MOVJ EC00441
SMOVL C00442 BC00442 V=1000.0  +MOVJ EC00442
SMOVL C00443 BC00443 V=1000.0  +MOVJ EC00443
SFTOF3D
MOVJ C00444 BC00444 VJ=100.00  +MOVJ EC00444 VJ=100.00
'Path W1876
SFTOF3D
SFTON3D P038
MOVJ C00445 BC00445 VJ=100.00  +MOVJ EC00445 VJ=100.00
MOVJ C00446 BC00446 VJ=100.00  +MOVJ EC00446 VJ=100.00
SMOVL C00447 BC00447 V=400.0  +MOVJ EC00447
SMOVL C00448 BC00448 V=100.0 PL=0  +MOVJ EC00448
SREFP 1 C00449 BC00449  +REFP EC00449
SREFP 2 C00450 BC00450  +REFP EC00450
MACRO1 MJ#(0) ARGF0
ARCON
SMOVL C00451 BC00451 V=10.0  +MOVJ EC00451
SMOVL C00452 BC00452 V=10.0  +MOVJ EC00452
ARCOF
SMOVL C00453 BC00453 V=400.0  +MOVJ EC00453
SMOVL C00454 BC00454 V=1000.0  +MOVJ EC00454
SFTOF3D
'Path W1877
SFTOF3D
SFTON3D P038
SMOVL C00455 BC00455 V=400.0  +MOVJ EC00455
SMOVL C00456 BC00456 V=100.0 PL=0  +MOVJ EC00456
SREFP 1 C00457 BC00457  +REFP EC00457
SREFP 2 C00458 BC00458  +REFP EC00458
MACRO1 MJ#(0) ARGF0
ARCON
SMOVL C00459 BC00459 V=10.0  +MOVJ EC00459
SMOVL C00460 BC00460 V=10.0  +MOVJ EC00460
SMOVL C00461 BC00461 V=10.0  +MOVJ EC00461
ARCOF
SMOVL C00462 BC00462 V=400.0  +MOVJ EC00462
SFTOF3D
MOVJ C00463 BC00463 VJ=100.00  +MOVJ EC00463 VJ=100.00
'Path W1878
SFTOF3D
SFTON3D P039
MOVJ C00464 BC00464 VJ=100.00  +MOVJ EC00464 VJ=100.00
MOVJ C00465 BC00465 VJ=100.00  +MOVJ EC00465 VJ=100.00
SMOVL C00466 BC00466 V=400.0  +MOVJ EC00466
SMOVL C00467 BC00467 V=100.0 PL=0  +MOVJ EC00467
SREFP 1 C00468 BC00468  +REFP EC00468
SREFP 2 C00469 BC00469  +REFP EC00469
MACRO1 MJ#(0) ARGF0
ARCON
SMOVL C00470 BC00470 V=10.0  +MOVJ EC00470
ARCOF
SMOVL C00471 BC00471 V=400.0  +MOVJ EC00471
SMOVL C00472 BC00472 V=1000.0  +MOVJ EC00472
SMOVL C00473 BC00473 V=1000.0  +MOVJ EC00473
SFTOF3D
'Path W1879
SFTOF3D
SFTON3D P042
MOVJ C00474 BC00474 VJ=100.00  +MOVJ EC00474 VJ=100.00
COMM MOVJ C00475 BC00475 VJ=100.00  +MOVJ EC00475 VJ=100.00
COMM SMOVL C00476 BC00476 V=400.0  +MOVJ EC00476
COMM SMOVL C00477 BC00477 V=100.0 PL=0  +MOVJ EC00477
COMM SREFP 1 C00478 BC00478  +REFP EC00478
COMM SREFP 2 C00479 BC00479  +REFP EC00479
COMM MACRO1 MJ#(0) ARGF0
COMM ARCON
COMM SMOVL C00480 BC00480 V=10.0  +MOVJ EC00480
COMM SMOVL C00481 BC00481 V=10.0  +MOVJ EC00481
COMM SMOVL C00482 BC00482 V=10.0  +MOVJ EC00482
COMM ARCOF
COMM SMOVL C00483 BC00483 V=400.0  +MOVJ EC00483
COMM SMOVL C00484 BC00484 V=1000.0  +MOVJ EC00484
SFTOF3D
'Path W1880
COMM SFTOF3D
COMM SFTON3D P041
COMM MOVJ C00485 BC00485 VJ=100.00  +MOVJ EC00485 VJ=100.00
COMM SMOVL C00486 BC00486 V=400.0  +MOVJ EC00486
COMM SMOVL C00487 BC00487 V=100.0 PL=0  +MOVJ EC00487
COMM SREFP 1 C00488 BC00488  +REFP EC00488
COMM SREFP 2 C00489 BC00489  +REFP EC00489
COMM MACRO1 MJ#(0) ARGF0
COMM ARCON
COMM SMOVL C00490 BC00490 V=10.0  +MOVJ EC00490
COMM ARCOF
COMM SMOVL C00491 BC00491 V=400.0  +MOVJ EC00491
COMM SMOVL C00492 BC00492 V=1000.0  +MOVJ EC00492
SFTOF3D
'Path W1881
COMM SFTOF3D
COMM SFTON3D P040
COMM MOVJ C00493 BC00493 VJ=100.00  +MOVJ EC00493 VJ=100.00
COMM SMOVL C00494 BC00494 V=400.0  +MOVJ EC00494
COMM SMOVL C00495 BC00495 V=100.0 PL=0  +MOVJ EC00495
COMM SREFP 1 C00496 BC00496  +REFP EC00496
COMM SREFP 2 C00497 BC00497  +REFP EC00497
COMM MACRO1 MJ#(0) ARGF0
COMM ARCON
COMM SMOVL C00498 BC00498 V=10.0  +MOVJ EC00498
COMM ARCOF
COMM SMOVL C00499 BC00499 V=400.0  +MOVJ EC00499
COMM SMOVL C00500 BC00500 V=1000.0  +MOVJ EC00500
COMM SMOVL C00501 BC00501 V=1000.0  +MOVJ EC00501
SFTOF3D
MOVJ C00502 BC00502 VJ=20.00  +MOVJ EC00502 VJ=20.00
'Path W1882
SFTOF3D
SFTON3D P043
MOVJ C00503 BC00503 VJ=100.00  +MOVJ EC00503 VJ=100.00
SMOVL C00504 BC00504 V=400.0  +MOVJ EC00504
SMOVL C00505 BC00505 V=100.0 PL=0  +MOVJ EC00505
SREFP 1 C00506 BC00506  +REFP EC00506
SREFP 2 C00507 BC00507  +REFP EC00507
MACRO1 MJ#(0) ARGF0
ARCON
COMM SMOVL C00508 BC00508 V=10.0  +MOVJ EC00508
COMM SMOVL C00509 BC00509 V=10.0  +MOVJ EC00509
COMM SMOVL C00510 BC00510 V=10.0  +MOVJ EC00510
COMM SMOVL C00511 BC00511 V=10.0  +MOVJ EC00511
COMM SMOVL C00512 BC00512 V=10.0  +MOVJ EC00512
COMM SMOVL C00513 BC00513 V=10.0  +MOVJ EC00513
COMM SMOVL C00514 BC00514 V=10.0  +MOVJ EC00514
SMOVL C00515 BC00515 V=10.0  +MOVJ EC00515
SMOVL C00516 BC00516 V=10.0  +MOVJ EC00516
SMOVL C00517 BC00517 V=10.0  +MOVJ EC00517
SMOVL C00518 BC00518 V=10.0  +MOVJ EC00518
SMOVL C00519 BC00519 V=10.0  +MOVJ EC00519
SMOVL C00520 BC00520 V=10.0  +MOVJ EC00520
SMOVL C00521 BC00521 V=10.0  +MOVJ EC00521
SMOVL C00522 BC00522 V=10.0  +MOVJ EC00522
ARCOF
SMOVL C00523 BC00523 V=400.0  +MOVJ EC00523
SMOVL C00524 BC00524 V=1000.0  +MOVJ EC00524
SFTOF3D
MOVJ C00525 BC00525 VJ=100.00  +MOVJ EC00525 VJ=100.00
MOVJ C00526 BC00526 VJ=100.00  +MOVJ EC00526 VJ=100.00
MOVJ C00527 BC00527 VJ=100.00  +MOVJ EC00527 VJ=100.00
*LABEL
'Down
MOVJ C00528 BC00528 VJ=50.00  +MOVJ EC00528 VJ=20.00
MOVJ C00529 BC00529 VJ=100.00  +MOVJ EC00529 VJ=100.00
MOVJ C00530 BC00530 VJ=100.00  +MOVJ EC00530 VJ=100.00
'1
'BRAKUJACY ELEMENT
'BRAKUJACY ELEMENT
'BRAKUJACY ELEMENT
'Path W1886
COMM SFTOF3D
COMM SFTON3D P023
COMM MOVJ C00531 BC00531 VJ=100.00  +MOVJ EC00531 VJ=100.00
COMM SMOVL C00532 BC00532 V=400.0  +MOVJ EC00532
